LIN {X 0,Y 467.559,Z 249.866,A -85,B 0,C 180,E1 -7501.046,E2 -7501.046} C_VEL
LIN {X 0,Y 467.576,Z 249.863,A -85,B 0,C 180,E1 -7504.243,E2 -7504.243} C_VEL
LIN {X 0,Y 467.538,Z 249.871,A -85,B 0,C 180,E1 -7507.188,E2 -7507.188} C_VEL
LIN {X 0,Y 467.588,Z 249.861,A -85,B 0,C 180,E1 -7510.263,E2 -7510.263} C_VEL
LIN {X 0,Y 467.605,Z 249.859,A -85,B 0,C 180,E1 -7512.572,E2 -7512.572} C_VEL
LIN {X 0,Y 467.561,Z 249.864,A -85,B 0,C 180,E1 -7516.177,E2 -7516.177} C_VEL
LIN {X 0,Y 467.577,Z 249.864,A -85,B 0,C 180,E1 -7518.722,E2 -7518.722} C_VEL
LIN {X 0,Y 467.565,Z 249.869,A -85,B 0,C 180,E1 -7521.407,E2 -7521.407} C_VEL
LIN {X 0,Y 467.55,Z 249.865,A -85,B 0,C 180,E1 -7524.261,E2 -7524.261} C_VEL
LIN {X 0,Y 467.569,Z 249.868,A -85,B 0,C 180,E1 -7527.322,E2 -7527.322} C_VEL
LIN {X 0,Y 467.566,Z 249.867,A -85,B 0,C 180,E1 -7530.666,E2 -7530.666} C_VEL
LIN {X 0,Y 467.616,Z 249.862,A -85,B 0,C 180,E1 -7533.201,E2 -7533.201} C_VEL
LIN {X 0,Y 467.581,Z 249.864,A -85,B 0,C 180,E1 -7536.469,E2 -7536.469} C_VEL
LIN {X 0,Y 467.612,Z 249.858,A -85,B 0,C 180,E1 -7539.778,E2 -7539.778} C_VEL
LIN {X 0,Y 467.599,Z 249.863,A -85,B 0,C 180,E1 -7542.508,E2 -7542.508} C_VEL
LIN {X 0,Y 467.596,Z 249.862,A -85,B 0,C 180,E1 -7545.198,E2 -7545.198} C_VEL
LIN {X 0,Y 467.645,Z 249.854,A -85,B 0,C 180,E1 -7547.856,E2 -7547.856} C_VEL
LIN {X 0,Y 467.672,Z 249.851,A -85,B 0,C 180,E1 -7551.358,E2 -7551.358} C_VEL
LIN {X 0,Y 467.738,Z 249.843,A -85,B 0,C 180,E1 -7553.964,E2 -7553.964} C_VEL
LIN {X 0,Y 467.852,Z 249.828,A -85,B 0,C 180,E1 -7557.418,E2 -7557.418} C_VEL
LIN {X 0,Y 467.874,Z 249.827,A -85,B 0,C 180,E1 -7560.001,E2 -7560.001} C_VEL
LIN {X 0,Y 467.852,Z 249.834,A -85,B 0,C 180,E1 -7562.584,E2 -7562.584} C_VEL
LIN {X 0,Y 467.736,Z 249.846,A -85,B 0,C 180,E1 -7566.039,E2 -7566.039} C_VEL
LIN {X 0,Y 467.675,Z 249.854,A -85,B 0,C 180,E1 -7568.644,E2 -7568.644} C_VEL
LIN {X 0,Y 467.649,Z 249.86,A -85,B 0,C 180,E1 -7572.147,E2 -7572.147} C_VEL
LIN {X 0,Y 467.661,Z 249.856,A -85,B 0,C 180,E1 -7575.894,E2 -7575.894} C_VEL
LIN {X 0,Y 467.618,Z 249.857,A -85,B 0,C 180,E1 -7579.309,E2 -7579.309} C_VEL
LIN {X 0,Y 467.53,Z 249.876,A -85,B 0,C 180,E1 -7582.075,E2 -7582.075} C_VEL
LIN {X 0,Y 467.599,Z 249.859,A -85,B 0,C 180,E1 -7584.888,E2 -7584.888} C_VEL
LIN {X 0,Y 467.617,Z 249.862,A -85,B 0,C 180,E1 -7587.77,E2 -7587.77} C_VEL
LIN {X 0,Y 467.569,Z 249.863,A -85,B 0,C 180,E1 -7591.047,E2 -7591.047} C_VEL
LIN {X 0,Y 467.587,Z 249.864,A -85,B 0,C 180,E1 -7594.244,E2 -7594.244} C_VEL
LIN {X 0,Y 467.548,Z 249.867,A -85,B 0,C 180,E1 -7597.188,E2 -7597.188} C_VEL
LIN {X 0,Y 467.576,Z 249.864,A -85,B 0,C 180,E1 -7600.266,E2 -7600.266} C_VEL
LIN {X 0,Y 467.585,Z 249.861,A -85,B 0,C 180,E1 -7602.568,E2 -7602.568} C_VEL
LIN {X 0,Y 467.569,Z 249.864,A -85,B 0,C 180,E1 -7605.054,E2 -7605.054} C_VEL
LIN {X 0,Y 467.589,Z 249.866,A -85,B 0,C 180,E1 -7607.441,E2 -7607.441} C_VEL
LIN {X 0,Y 467.559,Z 249.865,A -85,B 0,C 180,E1 -7610.854,E2 -7610.854} C_VEL
LIN {X 0,Y 467.56,Z 249.865,A -85,B 0,C 180,E1 -7614.262,E2 -7614.262} C_VEL
LIN {X 0,Y 467.583,Z 249.868,A -85,B 0,C 180,E1 -7617.322,E2 -7617.322} C_VEL
LIN {X 0,Y 467.571,Z 249.869,A -85,B 0,C 180,E1 -7620.668,E2 -7620.668} C_VEL
LIN {X 0,Y 467.657,Z 250.033,A -85,B 0,C 180,E1 -7622.276,E2 -7622.276} C_VEL
LIN {X 0,Y 470.699,Z 264.33,A -85,B 0,C 180,E1 -7624.816,E2 -7624.816} C_VEL
LIN {X 0,Y 470.515,Z 271.163,A -85,B 0,C 180,E1 -7625.927,E2 -7625.927} C_VEL
LIN {X 0,Y 469.617,Z 290.074,A -85,B 0,C 180,E1 -7628.951,E2 -7628.951} C_VEL
LIN {X 0,Y 469.483,Z 293.151,A -85,B 0,C 180,E1 -7629.44,E2 -7629.44} C_VEL
LIN {X 0,Y 473.262,Z 315.105,A -85,B 0,C 180,E1 -7629.948,E2 -7629.948} C_VEL
LIN {X 0,Y 472.112,Z 431.405,A -85,B 0,C 180,E1 -7631.756,E2 -7631.756} C_VEL
LIN {X 0,Y 471.636,Z 446.004,A -85,B 0,C 180,E1 -7632.157,E2 -7632.157} C_VEL
LIN {X 0,Y 471.213,Z 458.569,A -85,B 0,C 180,E1 -7632.659,E2 -7632.659} C_VEL
LIN {X 0,Y 470.615,Z 471.376,A -85,B 0,C 180,E1 -7633.332,E2 -7633.332} C_VEL
LIN {X 0,Y 469.961,Z 483.799,A -85,B 0,C 180,E1 -7634.162,E2 -7634.162} C_VEL
LIN {X 0,Y 469.293,Z 495.623,A -85,B 0,C 180,E1 -7635.14,E2 -7635.14} C_VEL
LIN {X 0,Y 468.67,Z 505.453,A -85,B 0,C 180,E1 -7636.118,E2 -7636.118} C_VEL
LIN {X 0,Y 468.146,Z 515.918,A -85,B 0,C 180,E1 -7637.373,E2 -7637.373} C_VEL
LIN {X 0,Y 467.67,Z 525.293,A -85,B 0,C 180,E1 -7638.734,E2 -7638.734} C_VEL
LIN {X 0,Y 467.228,Z 533.88,A -85,B 0,C 180,E1 -7640.258,E2 -7640.258} C_VEL
LIN {X 0,Y 466.947,Z 540.8,A -85,B 0,C 180,E1 -7641.78,E2 -7641.78} C_VEL
LIN {X 0,Y 466.824,Z 545.573,A -85,B 0,C 180,E1 -7643.083,E2 -7643.083} C_VEL
LIN {X 0,Y 466.728,Z 550.51,A -85,B 0,C 180,E1 -7644.816,E2 -7644.816} C_VEL
LIN {X 0,Y 466.652,Z 553.941,A -85,B 0,C 180,E1 -7646.546,E2 -7646.546} C_VEL
LIN {X 0,Y 466.605,Z 555.971,A -85,B 0,C 180,E1 -7648.274,E2 -7648.274} C_VEL
LIN {X 0,Y 466.598,Z 556.648,A -85,B 0,C 180,E1 -7650,E2 -7650} C_VEL
LIN {X 0,Y 466.605,Z 555.983,A -85,B 0,C 180,E1 -7651.726,E2 -7651.726} C_VEL
LIN {X 0,Y 466.652,Z 553.966,A -85,B 0,C 180,E1 -7653.454,E2 -7653.454} C_VEL
LIN {X 0,Y 466.729,Z 550.553,A -85,B 0,C 180,E1 -7655.183,E2 -7655.183} C_VEL
LIN {X 0,Y 466.823,Z 545.641,A -85,B 0,C 180,E1 -7656.917,E2 -7656.917} C_VEL
LIN {X 0,Y 467.027,Z 539.091,A -85,B 0,C 180,E1 -7658.655,E2 -7658.655} C_VEL
LIN {X 0,Y 467.299,Z 531.81,A -85,B 0,C 180,E1 -7660.178,E2 -7660.178} C_VEL
LIN {X 0,Y 467.852,Z 522.814,A -85,B 0,C 180,E1 -7661.7,E2 -7661.7} C_VEL
LIN {X 0,Y 468.33,Z 513.378,A -85,B 0,C 180,E1 -7663.008,E2 -7663.008} C_VEL
LIN {X 0,Y 468.972,Z 501.875,A -85,B 0,C 180,E1 -7664.315,E2 -7664.315} C_VEL
LIN {X 0,Y 469.736,Z 490.184,A -85,B 0,C 180,E1 -7665.4,E2 -7665.4} C_VEL
LIN {X 0,Y 470.352,Z 478.783,A -85,B 0,C 180,E1 -7666.269,E2 -7666.269} C_VEL
LIN {X 0,Y 471.025,Z 466.302,A -85,B 0,C 180,E1 -7667.034,E2 -7667.034} C_VEL
LIN {X 0,Y 471.6,Z 452.42,A -85,B 0,C 180,E1 -7667.692,E2 -7667.692} C_VEL
LIN {X 0,Y 472.176,Z 437.842,A -85,B 0,C 180,E1 -7668.183,E2 -7668.183} C_VEL
LIN {X 0,Y 472.478,Z 423.654,A -85,B 0,C 180,E1 -7668.482,E2 -7668.482} C_VEL
LIN {X 0,Y 473.578,Z 314.653,A -85,B 0,C 180,E1 -7670.174,E2 -7670.174} C_VEL
LIN {X 0,Y 469.645,Z 292.953,A -85,B 0,C 180,E1 -7670.718,E2 -7670.718} C_VEL
LIN {X 0,Y 470.739,Z 273.148,A -85,B 0,C 180,E1 -7673.94,E2 -7673.94} C_VEL
LIN {X 0,Y 471.057,Z 265.779,A -85,B 0,C 180,E1 -7675.163,E2 -7675.163} C_VEL
LIN {X 0,Y 468.784,Z 254.744,A -85,B 0,C 180,E1 -7677.196,E2 -7677.196} C_VEL
LIN {X 0,Y 467.611,Z 249.864,A -85,B 0,C 180,E1 -7678.134,E2 -7678.134} C_VEL
LIN {X 0,Y 467.583,Z 249.868,A -85,B 0,C 180,E1 -7681.739,E2 -7681.739} C_VEL
LIN {X 0,Y 467.564,Z 249.871,A -85,B 0,C 180,E1 -7684.832,E2 -7684.832} C_VEL
LIN {X 0,Y 467.564,Z 249.867,A -85,B 0,C 180,E1 -7688.044,E2 -7688.044} C_VEL
LIN {X 0,Y 467.582,Z 249.861,A -85,B 0,C 180,E1 -7691.276,E2 -7691.276} C_VEL
LIN {X 0,Y 467.573,Z 249.867,A -85,B 0,C 180,E1 -7693.822,E2 -7693.822} C_VEL
LIN {X 0,Y 467.586,Z 249.863,A -85,B 0,C 180,E1 -7697.439,E2 -7697.439} C_VEL
LIN {X 0,Y 467.579,Z 249.864,A -85,B 0,C 180,E1 -7700.854,E2 -7700.854} C_VEL
LIN {X 0,Y 467.559,Z 249.858,A -85,B 0,C 180,E1 -7704.259,E2 -7704.259} C_VEL
LIN {X 0,Y 467.578,Z 249.864,A -85,B 0,C 180,E1 -7707.32,E2 -7707.32} C_VEL
LIN {X 0,Y 467.572,Z 249.864,A -85,B 0,C 180,E1 -7710.665,E2 -7710.665} C_VEL
LIN {X 0,Y 467.611,Z 249.858,A -85,B 0,C 180,E1 -7713.198,E2 -7713.198} C_VEL
LIN {X 0,Y 467.587,Z 249.861,A -85,B 0,C 180,E1 -7716.467,E2 -7716.467} C_VEL
LIN {X 0,Y 467.616,Z 249.86,A -85,B 0,C 180,E1 -7719.776,E2 -7719.776} C_VEL
LIN {X 0,Y 467.602,Z 249.86,A -85,B 0,C 180,E1 -7722.506,E2 -7722.506} C_VEL
LIN {X 0,Y 467.599,Z 249.861,A -85,B 0,C 180,E1 -7725.195,E2 -7725.195} C_VEL
LIN {X 0,Y 467.649,Z 249.853,A -85,B 0,C 180,E1 -7727.853,E2 -7727.853} C_VEL
LIN {X 0,Y 467.674,Z 249.856,A -85,B 0,C 180,E1 -7731.356,E2 -7731.356} C_VEL
LIN {X 0,Y 467.735,Z 249.845,A -85,B 0,C 180,E1 -7733.961,E2 -7733.961} C_VEL
LIN {X 0,Y 467.851,Z 249.831,A -85,B 0,C 180,E1 -7737.416,E2 -7737.416} C_VEL
LIN {X 0,Y 467.872,Z 249.826,A -85,B 0,C 180,E1 -7739.999,E2 -7739.999} C_VEL
LIN {X 0,Y 467.85,Z 249.828,A -85,B 0,C 180,E1 -7742.582,E2 -7742.582} C_VEL
LIN {X 0,Y 467.733,Z 249.841,A -85,B 0,C 180,E1 -7746.036,E2 -7746.036} C_VEL
LIN {X 0,Y 467.671,Z 249.854,A -85,B 0,C 180,E1 -7748.642,E2 -7748.642} C_VEL
LIN {X 0,Y 467.645,Z 249.855,A -85,B 0,C 180,E1 -7752.144,E2 -7752.144} C_VEL
LIN {X 0,Y 467.626,Z 249.857,A -85,B 0,C 180,E1 -7755.694,E2 -7755.694} C_VEL
LIN {X 0,Y 467.605,Z 249.865,A -85,B 0,C 180,E1 -7758.764,E2 -7758.764} C_VEL
LIN {X 0,Y 467.597,Z 249.863,A -85,B 0,C 180,E1 -7761.277,E2 -7761.277} C_VEL
LIN {X 0,Y 467.562,Z 249.863,A -85,B 0,C 180,E1 -7763.942,E2 -7763.942} C_VEL
LIN {X 0,Y 467.603,Z 249.864,A -85,B 0,C 180,E1 -7766.799,E2 -7766.799} C_VEL
LIN {X 0,Y 467.573,Z 249.861,A -85,B 0,C 180,E1 -7769.735,E2 -7769.735} C_VEL
LIN {X 0,Y 467.569,Z 249.87,A -85,B 0,C 180,E1 -7772.758,E2 -7772.758} C_VEL
LIN {X 0,Y 467.541,Z 249.864,A -85,B 0,C 180,E1 -7775.889,E2 -7775.889} C_VEL
LIN {X 0,Y 467.601,Z 249.859,A -85,B 0,C 180,E1 -7779.141,E2 -7779.141} C_VEL
LIN {X 0,Y 467.604,Z 249.863,A -85,B 0,C 180,E1 -7782.571,E2 -7782.571} C_VEL
LIN {X 0,Y 467.559,Z 249.872,A -85,B 0,C 180,E1 -7786.176,E2 -7786.176} C_VEL
LIN {X 0,Y 467.574,Z 249.866,A -85,B 0,C 180,E1 -7788.721,E2 -7788.721} C_VEL
LIN {X 0,Y 467.606,Z 249.923,A -85,B 0,C 180,E1 -7791.4,E2 -7791.4} C_VEL
LIN {X 0,Y 470.158,Z 262.256,A -85,B 0,C 180,E1 -7793.981,E2 -7793.981} C_VEL
LIN {X 0,Y 469.866,Z 269.478,A -85,B 0,C 180,E1 -7795.349,E2 -7795.349} C_VEL
LIN {X 0,Y 473.76,Z 287.231,A -85,B 0,C 180,E1 -7795.831,E2 -7795.831} C_VEL
LIN {X 0,Y 472.595,Z 401.54,A -85,B 0,C 180,E1 -7797.615,E2 -7797.615} C_VEL
LIN {X 0,Y 472.256,Z 405.426,A -85,B 0,C 180,E1 -7797.674,E2 -7797.674} C_VEL
LIN {X 0,Y 470.929,Z 411.156,A -85,B 0,C 180,E1 -7797.757,E2 -7797.757} C_VEL
LIN {X 0,Y 466.084,Z 425.092,A -85,B 0,C 180,E1 -7798.009,E2 -7798.009} C_VEL
LIN {X 0,Y 465.031,Z 431.625,A -85,B 0,C 180,E1 -7798.248,E2 -7798.248} C_VEL
LIN {X 0,Y 464.439,Z 444.396,A -85,B 0,C 180,E1 -7798.911,E2 -7798.911} C_VEL
LIN {X 0,Y 463.798,Z 456.799,A -85,B 0,C 180,E1 -7799.734,E2 -7799.734} C_VEL
LIN {X 0,Y 463.03,Z 468.474,A -85,B 0,C 180,E1 -7800.693,E2 -7800.693} C_VEL
LIN {X 0,Y 462.274,Z 480.207,A -85,B 0,C 180,E1 -7801.882,E2 -7801.882} C_VEL
LIN {X 0,Y 461.648,Z 489.89,A -85,B 0,C 180,E1 -7803.071,E2 -7803.071} C_VEL
LIN {X 0,Y 461.034,Z 499.712,A -85,B 0,C 180,E1 -7804.534,E2 -7804.534} C_VEL
LIN {X 0,Y 460.527,Z 507.999,A -85,B 0,C 180,E1 -7806.047,E2 -7806.047} C_VEL
LIN {X 0,Y 460.144,Z 514.68,A -85,B 0,C 180,E1 -7807.553,E2 -7807.553} C_VEL
LIN {X 0,Y 459.849,Z 520.148,A -85,B 0,C 180,E1 -7809.095,E2 -7809.095} C_VEL
LIN {X 0,Y 459.686,Z 524.788,A -85,B 0,C 180,E1 -7810.81,E2 -7810.81} C_VEL
LIN {X 0,Y 459.553,Z 527.485,A -85,B 0,C 180,E1 -7812.19,E2 -7812.19} C_VEL
LIN {X 0,Y 459.45,Z 529.765,A -85,B 0,C 180,E1 -7814.018,E2 -7814.018} C_VEL
LIN {X 0,Y 459.494,Z 530.362,A -85,B 0,C 180,E1 -7814.929,E2 -7814.929} C_VEL
LIN {X 0,Y 459.43,Z 530.506,A -85,B 0,C 180,E1 -7816.735,E2 -7816.735} C_VEL
LIN {X 0,Y 459.553,Z 529.261,A -85,B 0,C 180,E1 -7818.533,E2 -7818.533} C_VEL
LIN {X 0,Y 459.528,Z 526.622,A -85,B 0,C 180,E1 -7820.315,E2 -7820.315} C_VEL
LIN {X 0,Y 459.759,Z 522.522,A -85,B 0,C 180,E1 -7822.093,E2 -7822.093} C_VEL
LIN {X 0,Y 459.989,Z 516.886,A -85,B 0,C 180,E1 -7823.861,E2 -7823.861} C_VEL
LIN {X 0,Y 460.24,Z 510.554,A -85,B 0,C 180,E1 -7825.402,E2 -7825.402} C_VEL
LIN {X 0,Y 460.669,Z 502.693,A -85,B 0,C 180,E1 -7826.939,E2 -7826.939} C_VEL
LIN {X 0,Y 461.204,Z 494.486,A -85,B 0,C 180,E1 -7828.254,E2 -7828.254} C_VEL
LIN {X 0,Y 461.807,Z 484.641,A -85,B 0,C 180,E1 -7829.564,E2 -7829.564} C_VEL
LIN {X 0,Y 462.521,Z 473.711,A -85,B 0,C 180,E1 -7830.762,E2 -7830.762} C_VEL
LIN {X 0,Y 463.251,Z 461.53,A -85,B 0,C 180,E1 -7831.848,E2 -7831.848} C_VEL
LIN {X 0,Y 463.921,Z 449.502,A -85,B 0,C 180,E1 -7832.713,E2 -7832.713} C_VEL
LIN {X 0,Y 464.518,Z 436.222,A -85,B 0,C 180,E1 -7833.47,E2 -7833.47} C_VEL
LIN {X 0,Y 464.988,Z 423.124,A -85,B 0,C 180,E1 -7834.036,E2 -7834.036} C_VEL
LIN {X 0,Y 465.325,Z 408.995,A -85,B 0,C 180,E1 -7834.467,E2 -7834.467} C_VEL
LIN {X 0,Y 465.621,Z 388.412,A -85,B 0,C 180,E1 -7834.833,E2 -7834.833} C_VEL
LIN {X 0,Y 466.608,Z 287.767,A -85,B 0,C 180,E1 -7836.404,E2 -7836.404} C_VEL
LIN {X 0,Y 462.682,Z 269.347,A -85,B 0,C 180,E1 -7836.879,E2 -7836.879} C_VEL
LIN {X 0,Y 462.829,Z 261.896,A -85,B 0,C 180,E1 -7838.294,E2 -7838.294} C_VEL
LIN {X 0,Y 460.594,Z 250.738,A -85,B 0,C 180,E1 -7840.606,E2 -7840.606} C_VEL
LIN {X 0,Y 460.578,Z 250.738,A -85,B 0,C 180,E1 -7843.231,E2 -7843.231} C_VEL
LIN {X 0,Y 460.586,Z 250.739,A -85,B 0,C 180,E1 -7845.998,E2 -7845.998} C_VEL
LIN {X 0,Y 460.557,Z 250.737,A -85,B 0,C 180,E1 -7848.902,E2 -7848.902} C_VEL
LIN {X 0,Y 460.502,Z 250.748,A -85,B 0,C 180,E1 -7851.486,E2 -7851.486} C_VEL
LIN {X 0,Y 460.533,Z 250.741,A -85,B 0,C 180,E1 -7854.332,E2 -7854.332} C_VEL
LIN {X 0,Y 460.57,Z 250.738,A -85,B 0,C 180,E1 -7857.243,E2 -7857.243} C_VEL
LIN {X 0,Y 460.513,Z 250.743,A -85,B 0,C 180,E1 -7860.239,E2 -7860.239} C_VEL
LIN {X 0,Y 460.515,Z 250.747,A -85,B 0,C 180,E1 -7863.325,E2 -7863.325} C_VEL
LIN {X 0,Y 460.465,Z 250.748,A -85,B 0,C 180,E1 -7866.53,E2 -7866.53} C_VEL
LIN {X 0,Y 460.571,Z 250.737,A -85,B 0,C 180,E1 -7869.857,E2 -7869.857} C_VEL
LIN {X 0,Y 460.529,Z 250.742,A -85,B 0,C 180,E1 -7872.905,E2 -7872.905} C_VEL
LIN {X 0,Y 460.51,Z 250.744,A -85,B 0,C 180,E1 -7875.829,E2 -7875.829} C_VEL
LIN {X 0,Y 460.53,Z 250.744,A -85,B 0,C 180,E1 -7878.991,E2 -7878.991} C_VEL
LIN {X 0,Y 460.534,Z 250.747,A -85,B 0,C 180,E1 -7881.27,E2 -7881.27} C_VEL
LIN {X 0,Y 460.501,Z 250.745,A -85,B 0,C 180,E1 -7884.556,E2 -7884.556} C_VEL
LIN {X 0,Y 460.52,Z 250.742,A -85,B 0,C 180,E1 -7887.717,E2 -7887.717} C_VEL
LIN {X 0,Y 460.535,Z 250.744,A -85,B 0,C 180,E1 -7890.771,E2 -7890.771} C_VEL
LIN {X 0,Y 460.556,Z 250.737,A -85,B 0,C 180,E1 -7893.736,E2 -7893.736} C_VEL
LIN {X 0,Y 460.534,Z 250.743,A -85,B 0,C 180,E1 -7896.625,E2 -7896.625} C_VEL
LIN {X 0,Y 460.54,Z 250.74,A -85,B 0,C 180,E1 -7899.454,E2 -7899.454} C_VEL
LIN {X 0,Y 460.548,Z 250.739,A -85,B 0,C 180,E1 -7902.231,E2 -7902.231} C_VEL
LIN {X 0,Y 460.555,Z 250.742,A -85,B 0,C 180,E1 -7904.966,E2 -7904.966} C_VEL
LIN {X 0,Y 460.598,Z 250.731,A -85,B 0,C 180,E1 -7907.667,E2 -7907.667} C_VEL
LIN {X 0,Y 460.619,Z 250.73,A -85,B 0,C 180,E1 -7911.225,E2 -7911.225} C_VEL
LIN {X 0,Y 460.704,Z 250.719,A -85,B 0,C 180,E1 -7913.871,E2 -7913.871} C_VEL
LIN {X 0,Y 460.817,Z 250.704,A -85,B 0,C 180,E1 -7917.379,E2 -7917.379} C_VEL
LIN {X 0,Y 460.845,Z 250.703,A -85,B 0,C 180,E1 -7920.001,E2 -7920.001} C_VEL
LIN {X 0,Y 460.817,Z 250.71,A -85,B 0,C 180,E1 -7922.624,E2 -7922.624} C_VEL
LIN {X 0,Y 460.702,Z 250.723,A -85,B 0,C 180,E1 -7926.131,E2 -7926.131} C_VEL
LIN {X 0,Y 460.622,Z 250.731,A -85,B 0,C 180,E1 -7928.777,E2 -7928.777} C_VEL
LIN {X 0,Y 460.607,Z 250.736,A -85,B 0,C 180,E1 -7932.446,E2 -7932.446} C_VEL
LIN {X 0,Y 460.617,Z 250.735,A -85,B 0,C 180,E1 -7936.008,E2 -7936.008} C_VEL
LIN {X 0,Y 460.564,Z 250.738,A -85,B 0,C 180,E1 -7939.617,E2 -7939.617} C_VEL
LIN {X 0,Y 460.506,Z 250.746,A -85,B 0,C 180,E1 -7942.43,E2 -7942.43} C_VEL
LIN {X 0,Y 460.564,Z 250.741,A -85,B 0,C 180,E1 -7945.803,E2 -7945.803} C_VEL
LIN {X 0,Y 460.551,Z 250.742,A -85,B 0,C 180,E1 -7948.234,E2 -7948.234} C_VEL
LIN {X 0,Y 460.521,Z 250.742,A -85,B 0,C 180,E1 -7951.285,E2 -7951.285} C_VEL
LIN {X 0,Y 460.531,Z 250.741,A -85,B 0,C 180,E1 -7954.507,E2 -7954.507} C_VEL
LIN {X 0,Y 460.526,Z 250.746,A -85,B 0,C 180,E1 -7957.622,E2 -7957.622} C_VEL
LIN {X 0,Y 460.54,Z 250.741,A -85,B 0,C 180,E1 -7960.27,E2 -7960.27} C_VEL
LIN {X 0,Y 460.498,Z 250.748,A -85,B 0,C 180,E1 -7963.376,E2 -7963.376} C_VEL
LIN {X 0,Y 460.499,Z 250.744,A -85,B 0,C 180,E1 -7966.626,E2 -7966.626} C_VEL
LIN {X 0,Y 460.538,Z 250.745,A -85,B 0,C 180,E1 -7969.732,E2 -7969.732} C_VEL
LIN {X 0,Y 460.499,Z 250.744,A -85,B 0,C 180,E1 -7972.525,E2 -7972.525} C_VEL
LIN {X 0,Y 460.547,Z 250.746,A -85,B 0,C 180,E1 -7975.625,E2 -7975.625} C_VEL
LIN {X 0,Y 460.539,Z 250.746,A -85,B 0,C 180,E1 -7978.745,E2 -7978.745} C_VEL
LIN {X 0,Y 460.584,Z 250.79,A -85,B 0,C 180,E1 -7982.015,E2 -7982.015} C_VEL
LIN {X 0,Y 463.706,Z 265.39,A -85,B 0,C 180,E1 -7984.65,E2 -7984.65} C_VEL
LIN {X 0,Y 463.848,Z 268.795,A -85,B 0,C 180,E1 -7985.224,E2 -7985.224} C_VEL
LIN {X 0,Y 462.711,Z 289.716,A -85,B 0,C 180,E1 -7988.622,E2 -7988.622} C_VEL
LIN {X 0,Y 462.617,Z 293.272,A -85,B 0,C 180,E1 -7989.156,E2 -7989.156} C_VEL
LIN {X 0,Y 466.496,Z 315.37,A -85,B 0,C 180,E1 -7989.675,E2 -7989.675} C_VEL
LIN {X 0,Y 465.322,Z 431.416,A -85,B 0,C 180,E1 -7991.508,E2 -7991.508} C_VEL
LIN {X 0,Y 464.838,Z 445.946,A -85,B 0,C 180,E1 -7991.916,E2 -7991.916} C_VEL
LIN {X 0,Y 464.346,Z 459.301,A -85,B 0,C 180,E1 -7992.464,E2 -7992.464} C_VEL
LIN {X 0,Y 463.691,Z 472.438,A -85,B 0,C 180,E1 -7993.178,E2 -7993.178} C_VEL
LIN {X 0,Y 462.981,Z 484.771,A -85,B 0,C 180,E1 -7994.03,E2 -7994.03} C_VEL
LIN {X 0,Y 462.303,Z 496.406,A -85,B 0,C 180,E1 -7995.023,E2 -7995.023} C_VEL
LIN {X 0,Y 461.593,Z 507.067,A -85,B 0,C 180,E1 -7996.125,E2 -7996.125} C_VEL
LIN {X 0,Y 461.075,Z 517.705,A -85,B 0,C 180,E1 -7997.462,E2 -7997.462} C_VEL
LIN {X 0,Y 460.57,Z 526.369,A -85,B 0,C 180,E1 -7998.781,E2 -7998.781} C_VEL
LIN {X 0,Y 460.129,Z 534.721,A -85,B 0,C 180,E1 -8000.328,E2 -8000.328} C_VEL
LIN {X 0,Y 459.889,Z 540.542,A -85,B 0,C 180,E1 -8001.652,E2 -8001.652} C_VEL
LIN {X 0,Y 459.734,Z 545.327,A -85,B 0,C 180,E1 -8002.975,E2 -8002.975} C_VEL
LIN {X 0,Y 459.638,Z 550.277,A -85,B 0,C 180,E1 -8004.736,E2 -8004.736} C_VEL
LIN {X 0,Y 459.549,Z 553.719,A -85,B 0,C 180,E1 -8006.493,E2 -8006.493} C_VEL
LIN {X 0,Y 459.518,Z 555.76,A -85,B 0,C 180,E1 -8008.247,E2 -8008.247} C_VEL
LIN {X 0,Y 459.529,Z 556.448,A -85,B 0,C 180,E1 -8010,E2 -8010} C_VEL
LIN {X 0,Y 459.518,Z 555.794,A -85,B 0,C 180,E1 -8011.753,E2 -8011.753} C_VEL
LIN {X 0,Y 459.548,Z 553.787,A -85,B 0,C 180,E1 -8013.507,E2 -8013.507} C_VEL
LIN {X 0,Y 459.643,Z 550.383,A -85,B 0,C 180,E1 -8015.264,E2 -8015.264} C_VEL
LIN {X 0,Y 459.734,Z 545.48,A -85,B 0,C 180,E1 -8017.024,E2 -8017.024} C_VEL
LIN {X 0,Y 459.96,Z 538.94,A -85,B 0,C 180,E1 -8018.789,E2 -8018.789} C_VEL
LIN {X 0,Y 460.271,Z 531.677,A -85,B 0,C 180,E1 -8020.335,E2 -8020.335} C_VEL
LIN {X 0,Y 460.84,Z 522.715,A -85,B 0,C 180,E1 -8021.881,E2 -8021.881} C_VEL
LIN {X 0,Y 461.349,Z 513.323,A -85,B 0,C 180,E1 -8023.209,E2 -8023.209} C_VEL
LIN {X 0,Y 461.987,Z 502.94,A -85,B 0,C 180,E1 -8024.424,E2 -8024.424} C_VEL
LIN {X 0,Y 462.788,Z 491.511,A -85,B 0,C 180,E1 -8025.524,E2 -8025.524} C_VEL
LIN {X 0,Y 463.536,Z 478.872,A -85,B 0,C 180,E1 -8026.515,E2 -8026.515} C_VEL
LIN {X 0,Y 464.215,Z 467.054,A -85,B 0,C 180,E1 -8027.258,E2 -8027.258} C_VEL
LIN {X 0,Y 464.816,Z 453.354,A -85,B 0,C 180,E1 -8027.931,E2 -8027.931} C_VEL
LIN {X 0,Y 465.43,Z 439.139,A -85,B 0,C 180,E1 -8028.43,E2 -8028.43} C_VEL
LIN {X 0,Y 465.814,Z 424.647,A -85,B 0,C 180,E1 -8028.756,E2 -8028.756} C_VEL
LIN {X 0,Y 466.883,Z 315.127,A -85,B 0,C 180,E1 -8030.491,E2 -8030.491} C_VEL
LIN {X 0,Y 463.077,Z 294.302,A -85,B 0,C 180,E1 -8031.027,E2 -8031.027} C_VEL
LIN {X 0,Y 462.808,Z 292.65,A -85,B 0,C 180,E1 -8031.084,E2 -8031.084} C_VEL
LIN {X 0,Y 463.969,Z 273.005,A -85,B 0,C 180,E1 -8034.337,E2 -8034.337} C_VEL
LIN {X 0,Y 464.196,Z 267.202,A -85,B 0,C 180,E1 -8035.322,E2 -8035.322} C_VEL
LIN {X 0,Y 461.48,Z 254.587,A -85,B 0,C 180,E1 -8037.703,E2 -8037.703} C_VEL
LIN {X 0,Y 460.575,Z 250.741,A -85,B 0,C 180,E1 -8038.479,E2 -8038.479} C_VEL
LIN {X 0,Y 460.521,Z 250.748,A -85,B 0,C 180,E1 -8041.282,E2 -8041.282} C_VEL
LIN {X 0,Y 460.531,Z 250.747,A -85,B 0,C 180,E1 -8044.504,E2 -8044.504} C_VEL
LIN {X 0,Y 460.5,Z 250.745,A -85,B 0,C 180,E1 -8047.622,E2 -8047.622} C_VEL
LIN {X 0,Y 460.541,Z 250.742,A -85,B 0,C 180,E1 -8050.268,E2 -8050.268} C_VEL
LIN {X 0,Y 460.523,Z 250.743,A -85,B 0,C 180,E1 -8053.371,E2 -8053.371} C_VEL
LIN {X 0,Y 460.497,Z 250.748,A -85,B 0,C 180,E1 -8056.623,E2 -8056.623} C_VEL
LIN {X 0,Y 460.539,Z 250.743,A -85,B 0,C 180,E1 -8059.729,E2 -8059.729} C_VEL
LIN {X 0,Y 460.497,Z 250.744,A -85,B 0,C 180,E1 -8062.522,E2 -8062.522} C_VEL
LIN {X 0,Y 460.544,Z 250.734,A -85,B 0,C 180,E1 -8065.623,E2 -8065.623} C_VEL
LIN {X 0,Y 460.533,Z 250.737,A -85,B 0,C 180,E1 -8068.743,E2 -8068.743} C_VEL
LIN {X 0,Y 460.55,Z 250.742,A -85,B 0,C 180,E1 -8071.766,E2 -8071.766} C_VEL
LIN {X 0,Y 460.553,Z 250.738,A -85,B 0,C 180,E1 -8074.704,E2 -8074.704} C_VEL
LIN {X 0,Y 460.505,Z 250.748,A -85,B 0,C 180,E1 -8077.57,E2 -8077.57} C_VEL
LIN {X 0,Y 460.562,Z 250.736,A -85,B 0,C 180,E1 -8080.383,E2 -8080.383} C_VEL
LIN {X 0,Y 460.559,Z 250.739,A -85,B 0,C 180,E1 -8083.145,E2 -8083.145} C_VEL
LIN {X 0,Y 460.548,Z 250.743,A -85,B 0,C 180,E1 -8085.867,E2 -8085.867} C_VEL
LIN {X 0,Y 460.605,Z 250.727,A -85,B 0,C 180,E1 -8088.558,E2 -8088.558} C_VEL
LIN {X 0,Y 460.687,Z 250.717,A -85,B 0,C 180,E1 -8092.107,E2 -8092.107} C_VEL
LIN {X 0,Y 460.689,Z 250.722,A -85,B 0,C 180,E1 -8094.747,E2 -8094.747} C_VEL
LIN {X 0,Y 460.816,Z 250.707,A -85,B 0,C 180,E1 -8097.376,E2 -8097.376} C_VEL
LIN {X 0,Y 460.843,Z 250.701,A -85,B 0,C 180,E1 -8099.999,E2 -8099.999} C_VEL
LIN {X 0,Y 460.815,Z 250.705,A -85,B 0,C 180,E1 -8102.621,E2 -8102.621} C_VEL
LIN {X 0,Y 460.699,Z 250.717,A -85,B 0,C 180,E1 -8106.129,E2 -8106.129} C_VEL
LIN {X 0,Y 460.618,Z 250.734,A -85,B 0,C 180,E1 -8108.775,E2 -8108.775} C_VEL
LIN {X 0,Y 460.601,Z 250.734,A -85,B 0,C 180,E1 -8112.444,E2 -8112.444} C_VEL
LIN {X 0,Y 460.588,Z 250.734,A -85,B 0,C 180,E1 -8115.997,E2 -8115.997} C_VEL
LIN {X 0,Y 460.558,Z 250.744,A -85,B 0,C 180,E1 -8118.901,E2 -8118.901} C_VEL
LIN {X 0,Y 460.548,Z 250.74,A -85,B 0,C 180,E1 -8121.482,E2 -8121.482} C_VEL
LIN {X 0,Y 460.531,Z 250.741,A -85,B 0,C 180,E1 -8124.331,E2 -8124.331} C_VEL
LIN {X 0,Y 460.559,Z 250.739,A -85,B 0,C 180,E1 -8127.243,E2 -8127.243} C_VEL
LIN {X 0,Y 460.512,Z 250.741,A -85,B 0,C 180,E1 -8130.238,E2 -8130.238} C_VEL
LIN {X 0,Y 460.515,Z 250.744,A -85,B 0,C 180,E1 -8133.324,E2 -8133.324} C_VEL
LIN {X 0,Y 460.464,Z 250.753,A -85,B 0,C 180,E1 -8136.529,E2 -8136.529} C_VEL
LIN {X 0,Y 460.561,Z 250.737,A -85,B 0,C 180,E1 -8139.857,E2 -8139.857} C_VEL
LIN {X 0,Y 460.528,Z 250.745,A -85,B 0,C 180,E1 -8142.904,E2 -8142.904} C_VEL
LIN {X 0,Y 460.509,Z 250.747,A -85,B 0,C 180,E1 -8145.828,E2 -8145.828} C_VEL
LIN {X 0,Y 460.527,Z 250.744,A -85,B 0,C 180,E1 -8148.99,E2 -8148.99} C_VEL
LIN {X 0,Y 460.578,Z 250.798,A -85,B 0,C 180,E1 -8151.094,E2 -8151.094} C_VEL
LIN {X 0,Y 463.119,Z 263.055,A -85,B 0,C 180,E1 -8153.713,E2 -8153.713} C_VEL
LIN {X 0,Y 463.209,Z 267.162,A -85,B 0,C 180,E1 -8154.526,E2 -8154.526} C_VEL
LIN {X 0,Y 463.049,Z 269.623,A -85,B 0,C 180,E1 -8154.997,E2 -8154.997} C_VEL
LIN {X 0,Y 467.2,Z 288.578,A -85,B 0,C 180,E1 -8155.526,E2 -8155.526} C_VEL
LIN {X 0,Y 465.834,Z 406.782,A -85,B 0,C 180,E1 -8157.418,E2 -8157.418} C_VEL
LIN {X 0,Y 465.445,Z 420.776,A -85,B 0,C 180,E1 -8157.817,E2 -8157.817} C_VEL
LIN {X 0,Y 465.031,Z 431.625,A -85,B 0,C 180,E1 -8158.248,E2 -8158.248} C_VEL
LIN {X 0,Y 464.152,Z 437.177,A -85,B 0,C 180,E1 -8158.477,E2 -8158.477} C_VEL
LIN {X 0,Y 460.955,Z 446.079,A -85,B 0,C 180,E1 -8158.853,E2 -8158.853} C_VEL
LIN {X 0,Y 457.735,Z 454.693,A -85,B 0,C 180,E1 -8159.315,E2 -8159.315} C_VEL
LIN {X 0,Y 456.823,Z 459.74,A -85,B 0,C 180,E1 -8159.674,E2 -8159.674} C_VEL
LIN {X 0,Y 456.035,Z 471.505,A -85,B 0,C 180,E1 -8160.706,E2 -8160.706} C_VEL
LIN {X 0,Y 455.274,Z 481.988,A -85,B 0,C 180,E1 -8161.824,E2 -8161.824} C_VEL
LIN {X 0,Y 454.61,Z 492.022,A -85,B 0,C 180,E1 -8163.117,E2 -8163.117} C_VEL
LIN {X 0,Y 453.973,Z 501.266,A -85,B 0,C 180,E1 -8164.559,E2 -8164.559} C_VEL
LIN {X 0,Y 453.45,Z 509.431,A -85,B 0,C 180,E1 -8166.121,E2 -8166.121} C_VEL
LIN {X 0,Y 453.049,Z 515.927,A -85,B 0,C 180,E1 -8167.663,E2 -8167.663} C_VEL
LIN {X 0,Y 452.77,Z 520.725,A -85,B 0,C 180,E1 -8169.084,E2 -8169.084} C_VEL
LIN {X 0,Y 452.614,Z 524.496,A -85,B 0,C 180,E1 -8170.498,E2 -8170.498} C_VEL
LIN {X 0,Y 452.483,Z 527.352,A -85,B 0,C 180,E1 -8171.903,E2 -8171.903} C_VEL
LIN {X 0,Y 452.358,Z 529.782,A -85,B 0,C 180,E1 -8173.761,E2 -8173.761} C_VEL
LIN {X 0,Y 452.411,Z 530.453,A -85,B 0,C 180,E1 -8174.688,E2 -8174.688} C_VEL
LIN {X 0,Y 452.342,Z 530.743,A -85,B 0,C 180,E1 -8176.524,E2 -8176.524} C_VEL
LIN {X 0,Y 452.454,Z 529.646,A -85,B 0,C 180,E1 -8178.351,E2 -8178.351} C_VEL
LIN {X 0,Y 452.433,Z 527.183,A -85,B 0,C 180,E1 -8180.162,E2 -8180.162} C_VEL
LIN {X 0,Y 452.659,Z 523.273,A -85,B 0,C 180,E1 -8181.968,E2 -8181.968} C_VEL
LIN {X 0,Y 452.895,Z 517.796,A -85,B 0,C 180,E1 -8183.764,E2 -8183.764} C_VEL
LIN {X 0,Y 453.117,Z 512.626,A -85,B 0,C 180,E1 -8185.107,E2 -8185.107} C_VEL
LIN {X 0,Y 453.511,Z 505.185,A -85,B 0,C 180,E1 -8186.669,E2 -8186.669} C_VEL
LIN {X 0,Y 454.027,Z 497.445,A -85,B 0,C 180,E1 -8188.004,E2 -8188.004} C_VEL
LIN {X 0,Y 454.639,Z 488.141,A -85,B 0,C 180,E1 -8189.336,E2 -8189.336} C_VEL
LIN {X 0,Y 455.331,Z 477.871,A -85,B 0,C 180,E1 -8190.553,E2 -8190.553} C_VEL
LIN {X 0,Y 456.09,Z 466.565,A -85,B 0,C 180,E1 -8191.656,E2 -8191.656} C_VEL
LIN {X 0,Y 456.836,Z 454.086,A -85,B 0,C 180,E1 -8192.645,E2 -8192.645} C_VEL
LIN {X 0,Y 457.448,Z 442.027,A -85,B 0,C 180,E1 -8193.413,E2 -8193.413} C_VEL
LIN {X 0,Y 458.03,Z 427.994,A -85,B 0,C 180,E1 -8194.103,E2 -8194.103} C_VEL
LIN {X 0,Y 458.462,Z 414.254,A -85,B 0,C 180,E1 -8194.589,E2 -8194.589} C_VEL
LIN {X 0,Y 458.753,Z 399.824,A -85,B 0,C 180,E1 -8194.916,E2 -8194.916} C_VEL
LIN {X 0,Y 459.919,Z 288.821,A -85,B 0,C 180,E1 -8196.672,E2 -8196.672} C_VEL
LIN {X 0,Y 455.756,Z 269.446,A -85,B 0,C 180,E1 -8197.198,E2 -8197.198} C_VEL
LIN {X 0,Y 455.879,Z 263.086,A -85,B 0,C 180,E1 -8198.421,E2 -8198.421} C_VEL
LIN {X 0,Y 453.547,Z 251.615,A -85,B 0,C 180,E1 -8200.829,E2 -8200.829} C_VEL
LIN {X 0,Y 453.524,Z 251.617,A -85,B 0,C 180,E1 -8203.441,E2 -8203.441} C_VEL
LIN {X 0,Y 453.531,Z 251.615,A -85,B 0,C 180,E1 -8206.196,E2 -8206.196} C_VEL
LIN {X 0,Y 453.506,Z 251.615,A -85,B 0,C 180,E1 -8209.041,E2 -8209.041} C_VEL
LIN {X 0,Y 453.463,Z 251.627,A -85,B 0,C 180,E1 -8211.836,E2 -8211.836} C_VEL
LIN {X 0,Y 453.511,Z 251.614,A -85,B 0,C 180,E1 -8214.734,E2 -8214.734} C_VEL
LIN {X 0,Y 453.525,Z 251.616,A -85,B 0,C 180,E1 -8217.962,E2 -8217.962} C_VEL
LIN {X 0,Y 453.469,Z 251.62,A -85,B 0,C 180,E1 -8220.759,E2 -8220.759} C_VEL
LIN {X 0,Y 453.464,Z 251.623,A -85,B 0,C 180,E1 -8223.913,E2 -8223.913} C_VEL
LIN {X 0,Y 453.458,Z 251.625,A -85,B 0,C 180,E1 -8227.188,E2 -8227.188} C_VEL
LIN {X 0,Y 453.523,Z 251.62,A -85,B 0,C 180,E1 -8229.445,E2 -8229.445} C_VEL
LIN {X 0,Y 453.479,Z 251.622,A -85,B 0,C 180,E1 -8232.992,E2 -8232.992} C_VEL
LIN {X 0,Y 453.463,Z 251.622,A -85,B 0,C 180,E1 -8235.781,E2 -8235.781} C_VEL
LIN {X 0,Y 453.483,Z 251.618,A -85,B 0,C 180,E1 -8238.212,E2 -8238.212} C_VEL
LIN {X 0,Y 453.519,Z 251.616,A -85,B 0,C 180,E1 -8240.788,E2 -8240.788} C_VEL
LIN {X 0,Y 453.444,Z 251.623,A -85,B 0,C 180,E1 -8243.918,E2 -8243.918} C_VEL
LIN {X 0,Y 453.47,Z 251.627,A -85,B 0,C 180,E1 -8247.152,E2 -8247.152} C_VEL
LIN {X 0,Y 453.502,Z 251.616,A -85,B 0,C 180,E1 -8250.272,E2 -8250.272} C_VEL
LIN {X 0,Y 453.502,Z 251.619,A -85,B 0,C 180,E1 -8253.295,E2 -8253.295} C_VEL
LIN {X 0,Y 453.492,Z 251.617,A -85,B 0,C 180,E1 -8256.24,E2 -8256.24} C_VEL
LIN {X 0,Y 453.472,Z 251.624,A -85,B 0,C 180,E1 -8259.119,E2 -8259.119} C_VEL
LIN {X 0,Y 453.501,Z 251.616,A -85,B 0,C 180,E1 -8261.946,E2 -8261.946} C_VEL
LIN {X 0,Y 453.529,Z 251.62,A -85,B 0,C 180,E1 -8264.727,E2 -8264.727} C_VEL
LIN {X 0,Y 453.553,Z 251.609,A -85,B 0,C 180,E1 -8267.472,E2 -8267.472} C_VEL
LIN {X 0,Y 453.583,Z 251.608,A -85,B 0,C 180,E1 -8271.088,E2 -8271.088} C_VEL
LIN {X 0,Y 453.671,Z 251.595,A -85,B 0,C 180,E1 -8273.776,E2 -8273.776} C_VEL
LIN {X 0,Y 453.758,Z 251.584,A -85,B 0,C 180,E1 -8277.338,E2 -8277.338} C_VEL
LIN {X 0,Y 453.815,Z 251.578,A -85,B 0,C 180,E1 -8280.001,E2 -8280.001} C_VEL
LIN {X 0,Y 453.758,Z 251.588,A -85,B 0,C 180,E1 -8282.664,E2 -8282.664} C_VEL
LIN {X 0,Y 453.67,Z 251.6,A -85,B 0,C 180,E1 -8286.227,E2 -8286.227} C_VEL
LIN {X 0,Y 453.586,Z 251.606,A -85,B 0,C 180,E1 -8288.915,E2 -8288.915} C_VEL
LIN {X 0,Y 453.557,Z 251.613,A -85,B 0,C 180,E1 -8292.53,E2 -8292.53} C_VEL
LIN {X 0,Y 453.551,Z 251.617,A -85,B 0,C 180,E1 -8296.197,E2 -8296.197} C_VEL
LIN {X 0,Y 453.515,Z 251.614,A -85,B 0,C 180,E1 -8299.042,E2 -8299.042} C_VEL
LIN {X 0,Y 453.472,Z 251.624,A -85,B 0,C 180,E1 -8301.837,E2 -8301.837} C_VEL
LIN {X 0,Y 453.51,Z 251.615,A -85,B 0,C 180,E1 -8304.736,E2 -8304.736} C_VEL
LIN {X 0,Y 453.53,Z 251.62,A -85,B 0,C 180,E1 -8307.961,E2 -8307.961} C_VEL
LIN {X 0,Y 453.48,Z 251.618,A -85,B 0,C 180,E1 -8310.76,E2 -8310.76} C_VEL
LIN {X 0,Y 453.475,Z 251.626,A -85,B 0,C 180,E1 -8313.914,E2 -8313.914} C_VEL
LIN {X 0,Y 453.468,Z 251.621,A -85,B 0,C 180,E1 -8317.189,E2 -8317.189} C_VEL
LIN {X 0,Y 453.515,Z 251.618,A -85,B 0,C 180,E1 -8319.448,E2 -8319.448} C_VEL
LIN {X 0,Y 453.462,Z 251.621,A -85,B 0,C 180,E1 -8322.996,E2 -8322.996} C_VEL
LIN {X 0,Y 453.465,Z 251.626,A -85,B 0,C 180,E1 -8325.78,E2 -8325.78} C_VEL
LIN {X 0,Y 453.479,Z 251.62,A -85,B 0,C 180,E1 -8328.21,E2 -8328.21} C_VEL
LIN {X 0,Y 453.471,Z 251.62,A -85,B 0,C 180,E1 -8330.798,E2 -8330.798} C_VEL
LIN {X 0,Y 453.454,Z 251.624,A -85,B 0,C 180,E1 -8333.918,E2 -8333.918} C_VEL
LIN {X 0,Y 453.484,Z 251.622,A -85,B 0,C 180,E1 -8337.152,E2 -8337.152} C_VEL
LIN {X 0,Y 453.476,Z 251.625,A -85,B 0,C 180,E1 -8340.269,E2 -8340.269} C_VEL
LIN {X 0,Y 453.554,Z 251.737,A -85,B 0,C 180,E1 -8341.783,E2 -8341.783} C_VEL
LIN {X 0,Y 456.924,Z 267.651,A -85,B 0,C 180,E1 -8344.696,E2 -8344.696} C_VEL
LIN {X 0,Y 456.157,Z 283.626,A -85,B 0,C 180,E1 -8347.346,E2 -8347.346} C_VEL
LIN {X 0,Y 455.661,Z 292.77,A -85,B 0,C 180,E1 -8348.844,E2 -8348.844} C_VEL
LIN {X 0,Y 459.794,Z 316.776,A -85,B 0,C 180,E1 -8349.418,E2 -8349.418} C_VEL
LIN {X 0,Y 458.546,Z 430.216,A -85,B 0,C 180,E1 -8351.225,E2 -8351.225} C_VEL
LIN {X 0,Y 458.077,Z 444.354,A -85,B 0,C 180,E1 -8351.611,E2 -8351.611} C_VEL
LIN {X 0,Y 457.523,Z 458.002,A -85,B 0,C 180,E1 -8352.162,E2 -8352.162} C_VEL
LIN {X 0,Y 456.847,Z 472.027,A -85,B 0,C 180,E1 -8352.929,E2 -8352.929} C_VEL
LIN {X 0,Y 456.108,Z 484.278,A -85,B 0,C 180,E1 -8353.783,E2 -8353.783} C_VEL
LIN {X 0,Y 455.397,Z 495.965,A -85,B 0,C 180,E1 -8354.79,E2 -8354.79} C_VEL
LIN {X 0,Y 454.632,Z 506.666,A -85,B 0,C 180,E1 -8355.909,E2 -8355.909} C_VEL
LIN {X 0,Y 454.073,Z 516.773,A -85,B 0,C 180,E1 -8357.188,E2 -8357.188} C_VEL
LIN {X 0,Y 453.553,Z 526.039,A -85,B 0,C 180,E1 -8358.605,E2 -8358.605} C_VEL
LIN {X 0,Y 453.061,Z 534.428,A -85,B 0,C 180,E1 -8360.175,E2 -8360.175} C_VEL
LIN {X 0,Y 452.814,Z 540.269,A -85,B 0,C 180,E1 -8361.521,E2 -8361.521} C_VEL
LIN {X 0,Y 452.658,Z 545.075,A -85,B 0,C 180,E1 -8362.865,E2 -8362.865} C_VEL
LIN {X 0,Y 452.549,Z 550.042,A -85,B 0,C 180,E1 -8364.654,E2 -8364.654} C_VEL
LIN {X 0,Y 452.448,Z 553.497,A -85,B 0,C 180,E1 -8366.438,E2 -8366.438} C_VEL
LIN {X 0,Y 452.501,Z 554.695,A -85,B 0,C 180,E1 -8367.329,E2 -8367.329} C_VEL
LIN {X 0,Y 452.427,Z 556.066,A -85,B 0,C 180,E1 -8369.11,E2 -8369.11} C_VEL
LIN {X 0,Y 452.427,Z 556.093,A -85,B 0,C 180,E1 -8370.89,E2 -8370.89} C_VEL
LIN {X 0,Y 452.501,Z 554.78,A -85,B 0,C 180,E1 -8372.67,E2 -8372.67} C_VEL
LIN {X 0,Y 452.472,Z 552.093,A -85,B 0,C 180,E1 -8374.454,E2 -8374.454} C_VEL
LIN {X 0,Y 452.585,Z 547.971,A -85,B 0,C 180,E1 -8376.24,E2 -8376.24} C_VEL
LIN {X 0,Y 452.742,Z 542.291,A -85,B 0,C 180,E1 -8378.031,E2 -8378.031} C_VEL
LIN {X 0,Y 453.049,Z 535.898,A -85,B 0,C 180,E1 -8379.599,E2 -8379.599} C_VEL
LIN {X 0,Y 453.525,Z 527.963,A -85,B 0,C 180,E1 -8381.169,E2 -8381.169} C_VEL
LIN {X 0,Y 454.033,Z 518.945,A -85,B 0,C 180,E1 -8382.627,E2 -8382.627} C_VEL
LIN {X 0,Y 454.649,Z 509.717,A -85,B 0,C 180,E1 -8383.863,E2 -8383.863} C_VEL
LIN {X 0,Y 455.39,Z 498.656,A -85,B 0,C 180,E1 -8385.095,E2 -8385.095} C_VEL
LIN {X 0,Y 456.291,Z 486.327,A -85,B 0,C 180,E1 -8386.21,E2 -8386.21} C_VEL
LIN {X 0,Y 457.071,Z 473.268,A -85,B 0,C 180,E1 -8387.159,E2 -8387.159} C_VEL
LIN {X 0,Y 457.856,Z 459.503,A -85,B 0,C 180,E1 -8387.936,E2 -8387.936} C_VEL
LIN {X 0,Y 458.493,Z 445.726,A -85,B 0,C 180,E1 -8388.516,E2 -8388.516} C_VEL
LIN {X 0,Y 458.975,Z 431.47,A -85,B 0,C 180,E1 -8388.931,E2 -8388.931} C_VEL
LIN {X 0,Y 459.763,Z 372.166,A -85,B 0,C 180,E1 -8389.904,E2 -8389.904} C_VEL
LIN {X 0,Y 460.281,Z 315.903,A -85,B 0,C 180,E1 -8390.813,E2 -8390.813} C_VEL
LIN {X 0,Y 456.68,Z 296.173,A -85,B 0,C 180,E1 -8391.333,E2 -8391.333} C_VEL
LIN {X 0,Y 455.972,Z 292.451,A -85,B 0,C 180,E1 -8391.449,E2 -8391.449} C_VEL
LIN {X 0,Y 457.235,Z 272.707,A -85,B 0,C 180,E1 -8394.779,E2 -8394.779} C_VEL
LIN {X 0,Y 457.304,Z 268.641,A -85,B 0,C 180,E1 -8395.487,E2 -8395.487} C_VEL
LIN {X 0,Y 454.946,Z 257.583,A -85,B 0,C 180,E1 -8397.608,E2 -8397.608} C_VEL
LIN {X 0,Y 453.509,Z 251.619,A -85,B 0,C 180,E1 -8398.838,E2 -8398.838} C_VEL
LIN {X 0,Y 453.465,Z 251.628,A -85,B 0,C 180,E1 -8401.798,E2 -8401.798} C_VEL
LIN {X 0,Y 453.48,Z 251.625,A -85,B 0,C 180,E1 -8404.988,E2 -8404.988} C_VEL
LIN {X 0,Y 453.463,Z 251.626,A -85,B 0,C 180,E1 -8408.311,E2 -8408.311} C_VEL
LIN {X 0,Y 453.494,Z 251.617,A -85,B 0,C 180,E1 -8410.608,E2 -8410.608} C_VEL
LIN {X 0,Y 453.48,Z 251.62,A -85,B 0,C 180,E1 -8413.246,E2 -8413.246} C_VEL
LIN {X 0,Y 453.464,Z 251.624,A -85,B 0,C 180,E1 -8415.778,E2 -8415.778} C_VEL
LIN {X 0,Y 453.477,Z 251.624,A -85,B 0,C 180,E1 -8418.208,E2 -8418.208} C_VEL
LIN {X 0,Y 453.491,Z 251.619,A -85,B 0,C 180,E1 -8420.792,E2 -8420.792} C_VEL
LIN {X 0,Y 453.453,Z 251.615,A -85,B 0,C 180,E1 -8423.916,E2 -8423.916} C_VEL
LIN {X 0,Y 453.479,Z 251.619,A -85,B 0,C 180,E1 -8427.15,E2 -8427.15} C_VEL
LIN {X 0,Y 453.51,Z 251.619,A -85,B 0,C 180,E1 -8430.27,E2 -8430.27} C_VEL
LIN {X 0,Y 453.501,Z 251.616,A -85,B 0,C 180,E1 -8433.293,E2 -8433.293} C_VEL
LIN {X 0,Y 453.498,Z 251.618,A -85,B 0,C 180,E1 -8436.238,E2 -8436.238} C_VEL
LIN {X 0,Y 453.476,Z 251.62,A -85,B 0,C 180,E1 -8439.116,E2 -8439.116} C_VEL
LIN {X 0,Y 453.505,Z 251.62,A -85,B 0,C 180,E1 -8441.943,E2 -8441.943} C_VEL
LIN {X 0,Y 453.532,Z 251.61,A -85,B 0,C 180,E1 -8444.725,E2 -8444.725} C_VEL
LIN {X 0,Y 453.554,Z 251.605,A -85,B 0,C 180,E1 -8448.378,E2 -8448.378} C_VEL
LIN {X 0,Y 453.644,Z 251.595,A -85,B 0,C 180,E1 -8451.984,E2 -8451.984} C_VEL
LIN {X 0,Y 453.663,Z 251.597,A -85,B 0,C 180,E1 -8454.666,E2 -8454.666} C_VEL
LIN {X 0,Y 453.756,Z 251.585,A -85,B 0,C 180,E1 -8457.336,E2 -8457.336} C_VEL
LIN {X 0,Y 453.814,Z 251.577,A -85,B 0,C 180,E1 -8459.999,E2 -8459.999} C_VEL
LIN {X 0,Y 453.756,Z 251.584,A -85,B 0,C 180,E1 -8462.662,E2 -8462.662} C_VEL
LIN {X 0,Y 453.666,Z 251.593,A -85,B 0,C 180,E1 -8466.224,E2 -8466.224} C_VEL
LIN {X 0,Y 453.582,Z 251.611,A -85,B 0,C 180,E1 -8468.912,E2 -8468.912} C_VEL
LIN {X 0,Y 453.552,Z 251.613,A -85,B 0,C 180,E1 -8472.528,E2 -8472.528} C_VEL
LIN {X 0,Y 453.532,Z 251.613,A -85,B 0,C 180,E1 -8476.195,E2 -8476.195} C_VEL
LIN {X 0,Y 453.508,Z 251.621,A -85,B 0,C 180,E1 -8479.04,E2 -8479.04} C_VEL
LIN {X 0,Y 453.485,Z 251.619,A -85,B 0,C 180,E1 -8481.834,E2 -8481.834} C_VEL
LIN {X 0,Y 453.502,Z 251.62,A -85,B 0,C 180,E1 -8484.733,E2 -8484.733} C_VEL
LIN {X 0,Y 453.52,Z 251.615,A -85,B 0,C 180,E1 -8487.959,E2 -8487.959} C_VEL
LIN {X 0,Y 453.469,Z 251.615,A -85,B 0,C 180,E1 -8490.758,E2 -8490.758} C_VEL
LIN {X 0,Y 453.463,Z 251.623,A -85,B 0,C 180,E1 -8493.912,E2 -8493.912} C_VEL
LIN {X 0,Y 453.457,Z 251.625,A -85,B 0,C 180,E1 -8497.187,E2 -8497.187} C_VEL
LIN {X 0,Y 453.517,Z 251.613,A -85,B 0,C 180,E1 -8499.445,E2 -8499.445} C_VEL
LIN {X 0,Y 453.477,Z 251.623,A -85,B 0,C 180,E1 -8502.991,E2 -8502.991} C_VEL
LIN {X 0,Y 453.462,Z 251.625,A -85,B 0,C 180,E1 -8505.78,E2 -8505.78} C_VEL
LIN {X 0,Y 453.481,Z 251.625,A -85,B 0,C 180,E1 -8508.211,E2 -8508.211} C_VEL
LIN {X 0,Y 453.534,Z 251.716,A -85,B 0,C 180,E1 -8510.784,E2 -8510.784} C_VEL
LIN {X 0,Y 455.95,Z 263.124,A -85,B 0,C 180,E1 -8513.273,E2 -8513.273} C_VEL
LIN {X 0,Y 456.404,Z 267.551,A -85,B 0,C 180,E1 -8514.188,E2 -8514.188} C_VEL
LIN {X 0,Y 456.287,Z 269.975,A -85,B 0,C 180,E1 -8514.638,E2 -8514.638} C_VEL
LIN {X 0,Y 460.485,Z 288.515,A -85,B 0,C 180,E1 -8515.177,E2 -8515.177} C_VEL
LIN {X 0,Y 460.561,Z 299.284,A -85,B 0,C 180,E1 -8515.361,E2 -8515.361} C_VEL
LIN {X 0,Y 459.225,Z 406.215,A -85,B 0,C 180,E1 -8517.091,E2 -8517.091} C_VEL
LIN {X 0,Y 458.826,Z 420.163,A -85,B 0,C 180,E1 -8517.484,E2 -8517.484} C_VEL
LIN {X 0,Y 458.255,Z 433.992,A -85,B 0,C 180,E1 -8518.056,E2 -8518.056} C_VEL
LIN {X 0,Y 457.603,Z 447.074,A -85,B 0,C 180,E1 -8518.78,E2 -8518.78} C_VEL
LIN {X 0,Y 456.823,Z 459.74,A -85,B 0,C 180,E1 -8519.674,E2 -8519.674} C_VEL
LIN {X 0,Y 455.905,Z 464.738,A -85,B 0,C 180,E1 -8520.058,E2 -8520.058} C_VEL
LIN {X 0,Y 452.617,Z 472.694,A -85,B 0,C 180,E1 -8520.677,E2 -8520.677} C_VEL
LIN {X 0,Y 449.255,Z 480.269,A -85,B 0,C 180,E1 -8521.369,E2 -8521.369} C_VEL
LIN {X 0,Y 448.235,Z 484.609,A -85,B 0,C 180,E1 -8521.863,E2 -8521.863} C_VEL
LIN {X 0,Y 447.597,Z 493.774,A -85,B 0,C 180,E1 -8523.107,E2 -8523.107} C_VEL
LIN {X 0,Y 446.905,Z 502.997,A -85,B 0,C 180,E1 -8524.626,E2 -8524.626} C_VEL
LIN {X 0,Y 446.448,Z 509.562,A -85,B 0,C 180,E1 -8525.924,E2 -8525.924} C_VEL
LIN {X 0,Y 446.056,Z 515.302,A -85,B 0,C 180,E1 -8527.294,E2 -8527.294} C_VEL
LIN {X 0,Y 445.751,Z 520.268,A -85,B 0,C 180,E1 -8528.739,E2 -8528.739} C_VEL
LIN {X 0,Y 445.577,Z 524.208,A -85,B 0,C 180,E1 -8530.178,E2 -8530.178} C_VEL
LIN {X 0,Y 445.427,Z 527.211,A -85,B 0,C 180,E1 -8531.606,E2 -8531.606} C_VEL
LIN {X 0,Y 445.268,Z 529.802,A -85,B 0,C 180,E1 -8533.495,E2 -8533.495} C_VEL
LIN {X 0,Y 445.311,Z 530.546,A -85,B 0,C 180,E1 -8534.437,E2 -8534.437} C_VEL
LIN {X 0,Y 445.254,Z 530.98,A -85,B 0,C 180,E1 -8536.305,E2 -8536.305} C_VEL
LIN {X 0,Y 445.369,Z 530.024,A -85,B 0,C 180,E1 -8538.163,E2 -8538.163} C_VEL
LIN {X 0,Y 445.346,Z 527.702,A -85,B 0,C 180,E1 -8540.004,E2 -8540.004} C_VEL
LIN {X 0,Y 445.558,Z 523.956,A -85,B 0,C 180,E1 -8541.839,E2 -8541.839} C_VEL
LIN {X 0,Y 445.804,Z 518.697,A -85,B 0,C 180,E1 -8543.665,E2 -8543.665} C_VEL
LIN {X 0,Y 446.016,Z 513.624,A -85,B 0,C 180,E1 -8545.028,E2 -8545.028} C_VEL
LIN {X 0,Y 446.436,Z 506.396,A -85,B 0,C 180,E1 -8546.616,E2 -8546.616} C_VEL
LIN {X 0,Y 447.036,Z 497.464,A -85,B 0,C 180,E1 -8548.198,E2 -8548.198} C_VEL
LIN {X 0,Y 447.71,Z 488.104,A -85,B 0,C 180,E1 -8549.55,E2 -8549.55} C_VEL
LIN {X 0,Y 448.478,Z 476.724,A -85,B 0,C 180,E1 -8550.898,E2 -8550.898} C_VEL
LIN {X 0,Y 449.29,Z 465.123,A -85,B 0,C 180,E1 -8552.017,E2 -8552.017} C_VEL
LIN {X 0,Y 450.086,Z 452.259,A -85,B 0,C 180,E1 -8553.021,E2 -8553.021} C_VEL
LIN {X 0,Y 450.722,Z 439.671,A -85,B 0,C 180,E1 -8553.8,E2 -8553.8} C_VEL
LIN {X 0,Y 451.356,Z 425.522,A -85,B 0,C 180,E1 -8554.465,E2 -8554.465} C_VEL
LIN {X 0,Y 451.737,Z 411.253,A -85,B 0,C 180,E1 -8554.937,E2 -8554.937} C_VEL
LIN {X 0,Y 452.016,Z 396.199,A -85,B 0,C 180,E1 -8555.241,E2 -8555.241} C_VEL
LIN {X 0,Y 453.25,Z 290.119,A -85,B 0,C 180,E1 -8556.941,E2 -8556.941} C_VEL
LIN {X 0,Y 448.85,Z 269.769,A -85,B 0,C 180,E1 -8557.478,E2 -8557.478} C_VEL
LIN {X 0,Y 449.071,Z 265.402,A -85,B 0,C 180,E1 -8558.323,E2 -8558.323} C_VEL
LIN {X 0,Y 446.545,Z 252.488,A -85,B 0,C 180,E1 -8561.059,E2 -8561.059} C_VEL
LIN {X 0,Y 446.473,Z 252.497,A -85,B 0,C 180,E1 -8563.657,E2 -8563.657} C_VEL
LIN {X 0,Y 446.476,Z 252.492,A -85,B 0,C 180,E1 -8566.459,E2 -8566.459} C_VEL
LIN {X 0,Y 446.455,Z 252.495,A -85,B 0,C 180,E1 -8569.303,E2 -8569.303} C_VEL
LIN {X 0,Y 446.404,Z 252.502,A -85,B 0,C 180,E1 -8572.2,E2 -8572.2} C_VEL
LIN {X 0,Y 446.457,Z 252.495,A -85,B 0,C 180,E1 -8575.152,E2 -8575.152} C_VEL
LIN {X 0,Y 446.47,Z 252.493,A -85,B 0,C 180,E1 -8578.179,E2 -8578.179} C_VEL
LIN {X 0,Y 446.417,Z 252.502,A -85,B 0,C 180,E1 -8581.3,E2 -8581.3} C_VEL
LIN {X 0,Y 446.416,Z 252.498,A -85,B 0,C 180,E1 -8584.523,E2 -8584.523} C_VEL
LIN {X 0,Y 446.425,Z 252.498,A -85,B 0,C 180,E1 -8588.084,E2 -8588.084} C_VEL
LIN {X 0,Y 446.434,Z 252.498,A -85,B 0,C 180,E1 -8590.921,E2 -8590.921} C_VEL
LIN {X 0,Y 446.432,Z 252.498,A -85,B 0,C 180,E1 -8593.841,E2 -8593.841} C_VEL
LIN {X 0,Y 446.433,Z 252.496,A -85,B 0,C 180,E1 -8596.398,E2 -8596.398} C_VEL
LIN {X 0,Y 446.456,Z 252.495,A -85,B 0,C 180,E1 -8599.806,E2 -8599.806} C_VEL
LIN {X 0,Y 446.421,Z 252.497,A -85,B 0,C 180,E1 -8602.125,E2 -8602.125} C_VEL
LIN {X 0,Y 446.418,Z 252.501,A -85,B 0,C 180,E1 -8605.478,E2 -8605.478} C_VEL
LIN {X 0,Y 446.407,Z 252.502,A -85,B 0,C 180,E1 -8608.701,E2 -8608.701} C_VEL
LIN {X 0,Y 446.472,Z 252.491,A -85,B 0,C 180,E1 -8611.822,E2 -8611.822} C_VEL
LIN {X 0,Y 446.447,Z 252.501,A -85,B 0,C 180,E1 -8614.849,E2 -8614.849} C_VEL
LIN {X 0,Y 446.437,Z 252.497,A -85,B 0,C 180,E1 -8618.246,E2 -8618.246} C_VEL
LIN {X 0,Y 446.446,Z 252.495,A -85,B 0,C 180,E1 -8621.65,E2 -8621.65} C_VEL
LIN {X 0,Y 446.497,Z 252.492,A -85,B 0,C 180,E1 -8624.481,E2 -8624.481} C_VEL
LIN {X 0,Y 446.506,Z 252.488,A -85,B 0,C 180,E1 -8627.385,E2 -8627.385} C_VEL
LIN {X 0,Y 446.529,Z 252.488,A -85,B 0,C 180,E1 -8630.946,E2 -8630.946} C_VEL
LIN {X 0,Y 446.639,Z 252.47,A -85,B 0,C 180,E1 -8633.678,E2 -8633.678} C_VEL
LIN {X 0,Y 446.702,Z 252.463,A -85,B 0,C 180,E1 -8637.296,E2 -8637.296} C_VEL
LIN {X 0,Y 446.785,Z 252.454,A -85,B 0,C 180,E1 -8640.001,E2 -8640.001} C_VEL
LIN {X 0,Y 446.702,Z 252.467,A -85,B 0,C 180,E1 -8642.706,E2 -8642.706} C_VEL
LIN {X 0,Y 446.639,Z 252.478,A -85,B 0,C 180,E1 -8646.325,E2 -8646.325} C_VEL
LIN {X 0,Y 446.531,Z 252.484,A -85,B 0,C 180,E1 -8649.057,E2 -8649.057} C_VEL
LIN {X 0,Y 446.516,Z 252.488,A -85,B 0,C 180,E1 -8652.731,E2 -8652.731} C_VEL
LIN {X 0,Y 446.514,Z 252.493,A -85,B 0,C 180,E1 -8656.239,E2 -8656.239} C_VEL
LIN {X 0,Y 446.464,Z 252.492,A -85,B 0,C 180,E1 -8659.304,E2 -8659.304} C_VEL
LIN {X 0,Y 446.414,Z 252.505,A -85,B 0,C 180,E1 -8662.201,E2 -8662.201} C_VEL
LIN {X 0,Y 446.453,Z 252.493,A -85,B 0,C 180,E1 -8665.154,E2 -8665.154} C_VEL
LIN {X 0,Y 446.481,Z 252.495,A -85,B 0,C 180,E1 -8668.18,E2 -8668.18} C_VEL
LIN {X 0,Y 446.417,Z 252.499,A -85,B 0,C 180,E1 -8671.301,E2 -8671.301} C_VEL
LIN {X 0,Y 446.428,Z 252.497,A -85,B 0,C 180,E1 -8674.524,E2 -8674.524} C_VEL
LIN {X 0,Y 446.429,Z 252.501,A -85,B 0,C 180,E1 -8678.083,E2 -8678.083} C_VEL
LIN {X 0,Y 446.425,Z 252.497,A -85,B 0,C 180,E1 -8680.919,E2 -8680.919} C_VEL
LIN {X 0,Y 446.401,Z 252.506,A -85,B 0,C 180,E1 -8683.847,E2 -8683.847} C_VEL
LIN {X 0,Y 446.399,Z 252.501,A -85,B 0,C 180,E1 -8686.404,E2 -8686.404} C_VEL
LIN {X 0,Y 446.426,Z 252.499,A -85,B 0,C 180,E1 -8689.083,E2 -8689.083} C_VEL
LIN {X 0,Y 446.407,Z 252.501,A -85,B 0,C 180,E1 -8692.122,E2 -8692.122} C_VEL
LIN {X 0,Y 446.43,Z 252.504,A -85,B 0,C 180,E1 -8695.478,E2 -8695.478} C_VEL
LIN {X 0,Y 446.417,Z 252.506,A -85,B 0,C 180,E1 -8698.7,E2 -8698.7} C_VEL
LIN {X 0,Y 446.511,Z 252.563,A -85,B 0,C 180,E1 -8701.523,E2 -8701.523} C_VEL
LIN {X 0,Y 450.028,Z 269.191,A -85,B 0,C 180,E1 -8704.617,E2 -8704.617} C_VEL
LIN {X 0,Y 449.205,Z 284.899,A -85,B 0,C 180,E1 -8707.259,E2 -8707.259} C_VEL
LIN {X 0,Y 448.743,Z 292.517,A -85,B 0,C 180,E1 -8708.526,E2 -8708.526} C_VEL
LIN {X 0,Y 453.044,Z 317.136,A -85,B 0,C 180,E1 -8709.136,E2 -8709.136} C_VEL
LIN {X 0,Y 451.76,Z 429.959,A -85,B 0,C 180,E1 -8710.961,E2 -8710.961} C_VEL
LIN {X 0,Y 451.281,Z 444.139,A -85,B 0,C 180,E1 -8711.353,E2 -8711.353} C_VEL
LIN {X 0,Y 450.661,Z 458.732,A -85,B 0,C 180,E1 -8711.958,E2 -8711.958} C_VEL
LIN {X 0,Y 449.933,Z 472.584,A -85,B 0,C 180,E1 -8712.736,E2 -8712.736} C_VEL
LIN {X 0,Y 449.148,Z 485.189,A -85,B 0,C 180,E1 -8713.641,E2 -8713.641} C_VEL
LIN {X 0,Y 448.293,Z 497.875,A -85,B 0,C 180,E1 -8714.776,E2 -8714.776} C_VEL
LIN {X 0,Y 447.551,Z 508.232,A -85,B 0,C 180,E1 -8715.913,E2 -8715.913} C_VEL
LIN {X 0,Y 447.012,Z 518.519,A -85,B 0,C 180,E1 -8717.285,E2 -8717.285} C_VEL
LIN {X 0,Y 446.452,Z 527.031,A -85,B 0,C 180,E1 -8718.652,E2 -8718.652} C_VEL
LIN {X 0,Y 445.966,Z 535.153,A -85,B 0,C 180,E1 -8720.247,E2 -8720.247} C_VEL
LIN {X 0,Y 445.661,Z 541.696,A -85,B 0,C 180,E1 -8721.841,E2 -8721.841} C_VEL
LIN {X 0,Y 445.541,Z 546.235,A -85,B 0,C 180,E1 -8723.206,E2 -8723.206} C_VEL
LIN {X 0,Y 445.461,Z 549.789,A -85,B 0,C 180,E1 -8724.568,E2 -8724.568} C_VEL
LIN {X 0,Y 445.348,Z 553.261,A -85,B 0,C 180,E1 -8726.381,E2 -8726.381} C_VEL
LIN {X 0,Y 445.425,Z 554.469,A -85,B 0,C 180,E1 -8727.287,E2 -8727.287} C_VEL
LIN {X 0,Y 445.337,Z 555.855,A -85,B 0,C 180,E1 -8729.096,E2 -8729.096} C_VEL
LIN {X 0,Y 445.337,Z 555.9,A -85,B 0,C 180,E1 -8730.904,E2 -8730.904} C_VEL
LIN {X 0,Y 445.425,Z 554.605,A -85,B 0,C 180,E1 -8732.713,E2 -8732.713} C_VEL
LIN {X 0,Y 445.394,Z 551.935,A -85,B 0,C 180,E1 -8734.525,E2 -8734.525} C_VEL
LIN {X 0,Y 445.512,Z 547.828,A -85,B 0,C 180,E1 -8736.34,E2 -8736.34} C_VEL
LIN {X 0,Y 445.687,Z 542.165,A -85,B 0,C 180,E1 -8738.159,E2 -8738.159} C_VEL
LIN {X 0,Y 446.006,Z 535.79,A -85,B 0,C 180,E1 -8739.752,E2 -8739.752} C_VEL
LIN {X 0,Y 446.501,Z 527.878,A -85,B 0,C 180,E1 -8741.347,E2 -8741.347} C_VEL
LIN {X 0,Y 447.009,Z 519.631,A -85,B 0,C 180,E1 -8742.715,E2 -8742.715} C_VEL
LIN {X 0,Y 447.718,Z 509.717,A -85,B 0,C 180,E1 -8744.082,E2 -8744.082} C_VEL
LIN {X 0,Y 448.511,Z 498.716,A -85,B 0,C 180,E1 -8745.332,E2 -8745.332} C_VEL
LIN {X 0,Y 449.479,Z 486.482,A -85,B 0,C 180,E1 -8746.463,E2 -8746.463} C_VEL
LIN {X 0,Y 450.292,Z 473.681,A -85,B 0,C 180,E1 -8747.414,E2 -8747.414} C_VEL
LIN {X 0,Y 451.13,Z 459.867,A -85,B 0,C 180,E1 -8748.212,E2 -8748.212} C_VEL
LIN {X 0,Y 451.785,Z 446.289,A -85,B 0,C 180,E1 -8748.802,E2 -8748.802} C_VEL
LIN {X 0,Y 452.291,Z 432.412,A -85,B 0,C 180,E1 -8749.221,E2 -8749.221} C_VEL
LIN {X 0,Y 452.782,Z 406.726,A -85,B 0,C 180,E1 -8749.671,E2 -8749.671} C_VEL
LIN {X 0,Y 453.721,Z 316.689,A -85,B 0,C 180,E1 -8751.144,E2 -8751.144} C_VEL
LIN {X 0,Y 449.931,Z 296.143,A -85,B 0,C 180,E1 -8751.703,E2 -8751.703} C_VEL
LIN {X 0,Y 449.127,Z 292.211,A -85,B 0,C 180,E1 -8751.835,E2 -8751.835} C_VEL
LIN {X 0,Y 450.404,Z 274.241,A -85,B 0,C 180,E1 -8754.916,E2 -8754.916} C_VEL
LIN {X 0,Y 450.39,Z 269.913,A -85,B 0,C 180,E1 -8755.689,E2 -8755.689} C_VEL
LIN {X 0,Y 448.036,Z 259.058,A -85,B 0,C 180,E1 -8757.817,E2 -8757.817} C_VEL
LIN {X 0,Y 446.495,Z 252.492,A -85,B 0,C 180,E1 -8759.175,E2 -8759.175} C_VEL
LIN {X 0,Y 446.423,Z 252.503,A -85,B 0,C 180,E1 -8762.361,E2 -8762.361} C_VEL
LIN {X 0,Y 446.419,Z 252.506,A -85,B 0,C 180,E1 -8765.625,E2 -8765.625} C_VEL
LIN {X 0,Y 446.443,Z 252.502,A -85,B 0,C 180,E1 -8769.026,E2 -8769.026} C_VEL
LIN {X 0,Y 446.45,Z 252.501,A -85,B 0,C 180,E1 -8772.279,E2 -8772.279} C_VEL
LIN {X 0,Y 446.453,Z 252.495,A -85,B 0,C 180,E1 -8775.102,E2 -8775.102} C_VEL
LIN {X 0,Y 446.425,Z 252.502,A -85,B 0,C 180,E1 -8778.608,E2 -8778.608} C_VEL
LIN {X 0,Y 446.441,Z 252.497,A -85,B 0,C 180,E1 -8780.972,E2 -8780.972} C_VEL
LIN {X 0,Y 446.417,Z 252.489,A -85,B 0,C 180,E1 -8784.373,E2 -8784.373} C_VEL
LIN {X 0,Y 446.419,Z 252.502,A -85,B 0,C 180,E1 -8787.637,E2 -8787.637} C_VEL
LIN {X 0,Y 446.464,Z 252.493,A -85,B 0,C 180,E1 -8790.791,E2 -8790.791} C_VEL
LIN {X 0,Y 446.473,Z 252.498,A -85,B 0,C 180,E1 -8793.847,E2 -8793.847} C_VEL
LIN {X 0,Y 446.423,Z 252.497,A -85,B 0,C 180,E1 -8796.822,E2 -8796.822} C_VEL
LIN {X 0,Y 446.437,Z 252.497,A -85,B 0,C 180,E1 -8799.736,E2 -8799.736} C_VEL
LIN {X 0,Y 446.457,Z 252.494,A -85,B 0,C 180,E1 -8802.596,E2 -8802.596} C_VEL
LIN {X 0,Y 446.463,Z 252.496,A -85,B 0,C 180,E1 -8805.411,E2 -8805.411} C_VEL
LIN {X 0,Y 446.511,Z 252.483,A -85,B 0,C 180,E1 -8808.192,E2 -8808.192} C_VEL
LIN {X 0,Y 446.592,Z 252.475,A -85,B 0,C 180,E1 -8811.857,E2 -8811.857} C_VEL
LIN {X 0,Y 446.637,Z 252.472,A -85,B 0,C 180,E1 -8814.581,E2 -8814.581} C_VEL
LIN {X 0,Y 446.7,Z 252.464,A -85,B 0,C 180,E1 -8817.293,E2 -8817.293} C_VEL
LIN {X 0,Y 446.784,Z 252.453,A -85,B 0,C 180,E1 -8819.999,E2 -8819.999} C_VEL
LIN {X 0,Y 446.7,Z 252.464,A -85,B 0,C 180,E1 -8822.704,E2 -8822.704} C_VEL
LIN {X 0,Y 446.636,Z 252.469,A -85,B 0,C 180,E1 -8826.323,E2 -8826.323} C_VEL
LIN {X 0,Y 446.528,Z 252.487,A -85,B 0,C 180,E1 -8829.054,E2 -8829.054} C_VEL
LIN {X 0,Y 446.51,Z 252.492,A -85,B 0,C 180,E1 -8832.729,E2 -8832.729} C_VEL
LIN {X 0,Y 446.484,Z 252.492,A -85,B 0,C 180,E1 -8836.227,E2 -8836.227} C_VEL
LIN {X 0,Y 446.458,Z 252.496,A -85,B 0,C 180,E1 -8839.302,E2 -8839.302} C_VEL
LIN {X 0,Y 446.42,Z 252.5,A -85,B 0,C 180,E1 -8842.198,E2 -8842.198} C_VEL
LIN {X 0,Y 446.445,Z 252.499,A -85,B 0,C 180,E1 -8845.151,E2 -8845.151} C_VEL
LIN {X 0,Y 446.471,Z 252.495,A -85,B 0,C 180,E1 -8848.178,E2 -8848.178} C_VEL
LIN {X 0,Y 446.405,Z 252.497,A -85,B 0,C 180,E1 -8851.299,E2 -8851.299} C_VEL
LIN {X 0,Y 446.416,Z 252.497,A -85,B 0,C 180,E1 -8854.522,E2 -8854.522} C_VEL
LIN {X 0,Y 446.423,Z 252.503,A -85,B 0,C 180,E1 -8858.082,E2 -8858.082} C_VEL
LIN {X 0,Y 446.433,Z 252.5,A -85,B 0,C 180,E1 -8860.92,E2 -8860.92} C_VEL
LIN {X 0,Y 446.43,Z 252.502,A -85,B 0,C 180,E1 -8863.84,E2 -8863.84} C_VEL
LIN {X 0,Y 446.432,Z 252.503,A -85,B 0,C 180,E1 -8866.396,E2 -8866.396} C_VEL
LIN {X 0,Y 446.456,Z 252.502,A -85,B 0,C 180,E1 -8869.805,E2 -8869.805} C_VEL
LIN {X 0,Y 446.501,Z 252.66,A -85,B 0,C 180,E1 -8870.465,E2 -8870.465} C_VEL
LIN {X 0,Y 449.051,Z 264.63,A -85,B 0,C 180,E1 -8873.129,E2 -8873.129} C_VEL
LIN {X 0,Y 449.546,Z 268.977,A -85,B 0,C 180,E1 -8874.047,E2 -8874.047} C_VEL
LIN {X 0,Y 449.466,Z 270.02,A -85,B 0,C 180,E1 -8874.253,E2 -8874.253} C_VEL
LIN {X 0,Y 453.864,Z 289.061,A -85,B 0,C 180,E1 -8874.829,E2 -8874.829} C_VEL
LIN {X 0,Y 454.137,Z 293.313,A -85,B 0,C 180,E1 -8874.917,E2 -8874.917} C_VEL
LIN {X 0,Y 452.592,Z 406.939,A -85,B 0,C 180,E1 -8876.786,E2 -8876.786} C_VEL
LIN {X 0,Y 452.163,Z 421.356,A -85,B 0,C 180,E1 -8877.21,E2 -8877.21} C_VEL
LIN {X 0,Y 451.538,Z 434.91,A -85,B 0,C 180,E1 -8877.787,E2 -8877.787} C_VEL
LIN {X 0,Y 450.875,Z 447.839,A -85,B 0,C 180,E1 -8878.522,E2 -8878.522} C_VEL
LIN {X 0,Y 450.032,Z 460.547,A -85,B 0,C 180,E1 -8879.44,E2 -8879.44} C_VEL
LIN {X 0,Y 449.215,Z 472.076,A -85,B 0,C 180,E1 -8880.475,E2 -8880.475} C_VEL
LIN {X 0,Y 448.426,Z 482.325,A -85,B 0,C 180,E1 -8881.589,E2 -8881.589} C_VEL
LIN {X 0,Y 448.235,Z 484.609,A -85,B 0,C 180,E1 -8881.863,E2 -8881.863} C_VEL
LIN {X 0,Y 447.236,Z 488.865,A -85,B 0,C 180,E1 -8882.384,E2 -8882.384} C_VEL
LIN {X 0,Y 443.929,Z 495.474,A -85,B 0,C 180,E1 -8883.236,E2 -8883.236} C_VEL
LIN {X 0,Y 440.697,Z 501.63,A -85,B 0,C 180,E1 -8884.15,E2 -8884.15} C_VEL
LIN {X 0,Y 439.817,Z 505.027,A -85,B 0,C 180,E1 -8884.76,E2 -8884.76} C_VEL
LIN {X 0,Y 439.239,Z 512.75,A -85,B 0,C 180,E1 -8886.422,E2 -8886.422} C_VEL
LIN {X 0,Y 438.876,Z 518.229,A -85,B 0,C 180,E1 -8887.89,E2 -8887.89} C_VEL
LIN {X 0,Y 438.591,Z 522.652,A -85,B 0,C 180,E1 -8889.359,E2 -8889.359} C_VEL
LIN {X 0,Y 438.419,Z 526.521,A -85,B 0,C 180,E1 -8891.042,E2 -8891.042} C_VEL
LIN {X 0,Y 438.247,Z 528.597,A -85,B 0,C 180,E1 -8892.261,E2 -8892.261} C_VEL
LIN {X 0,Y 438.229,Z 530.647,A -85,B 0,C 180,E1 -8894.197,E2 -8894.197} C_VEL
LIN {X 0,Y 438.154,Z 531.217,A -85,B 0,C 180,E1 -8896.078,E2 -8896.078} C_VEL
LIN {X 0,Y 438.255,Z 530.366,A -85,B 0,C 180,E1 -8898.009,E2 -8898.009} C_VEL
LIN {X 0,Y 438.265,Z 528.219,A -85,B 0,C 180,E1 -8899.84,E2 -8899.84} C_VEL
LIN {X 0,Y 438.469,Z 524.617,A -85,B 0,C 180,E1 -8901.706,E2 -8901.706} C_VEL
LIN {X 0,Y 438.688,Z 519.523,A -85,B 0,C 180,E1 -8903.561,E2 -8903.561} C_VEL
LIN {X 0,Y 438.905,Z 514.598,A -85,B 0,C 180,E1 -8904.948,E2 -8904.948} C_VEL
LIN {X 0,Y 439.357,Z 507.537,A -85,B 0,C 180,E1 -8906.561,E2 -8906.561} C_VEL
LIN {X 0,Y 439.958,Z 498.828,A -85,B 0,C 180,E1 -8908.169,E2 -8908.169} C_VEL
LIN {X 0,Y 440.623,Z 489.729,A -85,B 0,C 180,E1 -8909.543,E2 -8909.543} C_VEL
LIN {X 0,Y 441.448,Z 478.701,A -85,B 0,C 180,E1 -8910.912,E2 -8910.912} C_VEL
LIN {X 0,Y 442.295,Z 467.46,A -85,B 0,C 180,E1 -8912.049,E2 -8912.049} C_VEL
LIN {X 0,Y 443.093,Z 455.078,A -85,B 0,C 180,E1 -8913.069,E2 -8913.069} C_VEL
LIN {X 0,Y 443.824,Z 441.612,A -85,B 0,C 180,E1 -8913.949,E2 -8913.949} C_VEL
LIN {X 0,Y 444.409,Z 428.507,A -85,B 0,C 180,E1 -8914.606,E2 -8914.606} C_VEL
LIN {X 0,Y 444.911,Z 414.177,A -85,B 0,C 180,E1 -8915.126,E2 -8915.126} C_VEL
LIN {X 0,Y 445.213,Z 399.421,A -85,B 0,C 180,E1 -8915.463,E2 -8915.463} C_VEL
LIN {X 0,Y 446.546,Z 291.875,A -85,B 0,C 180,E1 -8917.209,E2 -8917.209} C_VEL
LIN {X 0,Y 442.711,Z 273.448,A -85,B 0,C 180,E1 -8917.695,E2 -8917.695} C_VEL
LIN {X 0,Y 442.012,Z 269.817,A -85,B 0,C 180,E1 -8917.816,E2 -8917.816} C_VEL
LIN {X 0,Y 441.925,Z 265.46,A -85,B 0,C 180,E1 -8918.689,E2 -8918.689} C_VEL
LIN {X 0,Y 439.517,Z 253.365,A -85,B 0,C 180,E1 -8921.296,E2 -8921.296} C_VEL
LIN {X 0,Y 439.424,Z 253.377,A -85,B 0,C 180,E1 -8923.881,E2 -8923.881} C_VEL
LIN {X 0,Y 439.436,Z 253.368,A -85,B 0,C 180,E1 -8926.731,E2 -8926.731} C_VEL
LIN {X 0,Y 439.417,Z 253.376,A -85,B 0,C 180,E1 -8929.625,E2 -8929.625} C_VEL
LIN {X 0,Y 439.351,Z 253.378,A -85,B 0,C 180,E1 -8932.576,E2 -8932.576} C_VEL
LIN {X 0,Y 439.4,Z 253.379,A -85,B 0,C 180,E1 -8935.585,E2 -8935.585} C_VEL
LIN {X 0,Y 439.411,Z 253.371,A -85,B 0,C 180,E1 -8938.673,E2 -8938.673} C_VEL
LIN {X 0,Y 439.369,Z 253.378,A -85,B 0,C 180,E1 -8942.034,E2 -8942.034} C_VEL
LIN {X 0,Y 439.382,Z 253.38,A -85,B 0,C 180,E1 -8945.341,E2 -8945.341} C_VEL
LIN {X 0,Y 439.387,Z 253.374,A -85,B 0,C 180,E1 -8948.594,E2 -8948.594} C_VEL
LIN {X 0,Y 439.392,Z 253.379,A -85,B 0,C 180,E1 -8951.26,E2 -8951.26} C_VEL
LIN {X 0,Y 439.396,Z 253.374,A -85,B 0,C 180,E1 -8954.729,E2 -8954.729} C_VEL
LIN {X 0,Y 439.399,Z 253.374,A -85,B 0,C 180,E1 -8957.798,E2 -8957.798} C_VEL
LIN {X 0,Y 439.439,Z 253.367,A -85,B 0,C 180,E1 -8960.231,E2 -8960.231} C_VEL
LIN {X 0,Y 439.365,Z 253.378,A -85,B 0,C 180,E1 -8963.714,E2 -8963.714} C_VEL
LIN {X 0,Y 439.361,Z 253.384,A -85,B 0,C 180,E1 -8967.055,E2 -8967.055} C_VEL
LIN {X 0,Y 439.384,Z 253.374,A -85,B 0,C 180,E1 -8970.276,E2 -8970.276} C_VEL
LIN {X 0,Y 439.422,Z 253.371,A -85,B 0,C 180,E1 -8973.59,E2 -8973.59} C_VEL
LIN {X 0,Y 439.375,Z 253.377,A -85,B 0,C 180,E1 -8976.431,E2 -8976.431} C_VEL
LIN {X 0,Y 439.377,Z 253.377,A -85,B 0,C 180,E1 -8979.398,E2 -8979.398} C_VEL
LIN {X 0,Y 439.421,Z 253.371,A -85,B 0,C 180,E1 -8982.311,E2 -8982.311} C_VEL
LIN {X 0,Y 439.439,Z 253.37,A -85,B 0,C 180,E1 -8985.175,E2 -8985.175} C_VEL
LIN {X 0,Y 439.474,Z 253.364,A -85,B 0,C 180,E1 -8988.002,E2 -8988.002} C_VEL
LIN {X 0,Y 439.539,Z 253.355,A -85,B 0,C 180,E1 -8991.727,E2 -8991.727} C_VEL
LIN {X 0,Y 439.615,Z 253.352,A -85,B 0,C 180,E1 -8994.497,E2 -8994.497} C_VEL
LIN {X 0,Y 439.628,Z 253.347,A -85,B 0,C 180,E1 -8998.169,E2 -8998.169} C_VEL
LIN {X 0,Y 439.755,Z 253.33,A -85,B 0,C 180,E1 -9000.001,E2 -9000.001} C_VEL
LIN {X 0,Y 439.649,Z 253.345,A -85,B 0,C 180,E1 -9002.75,E2 -9002.75} C_VEL
LIN {X 0,Y 439.611,Z 253.353,A -85,B 0,C 180,E1 -9006.426,E2 -9006.426} C_VEL
LIN {X 0,Y 439.493,Z 253.361,A -85,B 0,C 180,E1 -9009.203,E2 -9009.203} C_VEL
LIN {X 0,Y 439.46,Z 253.365,A -85,B 0,C 180,E1 -9012.939,E2 -9012.939} C_VEL
LIN {X 0,Y 439.455,Z 253.371,A -85,B 0,C 180,E1 -9016.356,E2 -9016.356} C_VEL
LIN {X 0,Y 439.398,Z 253.374,A -85,B 0,C 180,E1 -9019.628,E2 -9019.628} C_VEL
LIN {X 0,Y 439.361,Z 253.379,A -85,B 0,C 180,E1 -9022.577,E2 -9022.577} C_VEL
LIN {X 0,Y 439.401,Z 253.374,A -85,B 0,C 180,E1 -9025.586,E2 -9025.586} C_VEL
LIN {X 0,Y 439.422,Z 253.37,A -85,B 0,C 180,E1 -9028.674,E2 -9028.674} C_VEL
LIN {X 0,Y 439.38,Z 253.381,A -85,B 0,C 180,E1 -9032.034,E2 -9032.034} C_VEL
LIN {X 0,Y 439.394,Z 253.375,A -85,B 0,C 180,E1 -9035.342,E2 -9035.342} C_VEL
LIN {X 0,Y 439.388,Z 253.374,A -85,B 0,C 180,E1 -9038.595,E2 -9038.595} C_VEL
LIN {X 0,Y 439.387,Z 253.376,A -85,B 0,C 180,E1 -9041.258,E2 -9041.258} C_VEL
LIN {X 0,Y 439.401,Z 253.372,A -85,B 0,C 180,E1 -9044.73,E2 -9044.73} C_VEL
LIN {X 0,Y 439.396,Z 253.378,A -85,B 0,C 180,E1 -9047.797,E2 -9047.797} C_VEL
LIN {X 0,Y 439.389,Z 253.374,A -85,B 0,C 180,E1 -9050.224,E2 -9050.224} C_VEL
LIN {X 0,Y 439.374,Z 253.38,A -85,B 0,C 180,E1 -9053.714,E2 -9053.714} C_VEL
LIN {X 0,Y 439.374,Z 253.378,A -85,B 0,C 180,E1 -9057.055,E2 -9057.055} C_VEL
LIN {X 0,Y 439.42,Z 253.377,A -85,B 0,C 180,E1 -9060.804,E2 -9060.804} C_VEL
LIN {X 0,Y 439.457,Z 253.425,A -85,B 0,C 180,E1 -9061.265,E2 -9061.265} C_VEL
LIN {X 0,Y 442.675,Z 268.443,A -85,B 0,C 180,E1 -9064.114,E2 -9064.114} C_VEL
LIN {X 0,Y 443.087,Z 272.455,A -85,B 0,C 180,E1 -9064.837,E2 -9064.837} C_VEL
LIN {X 0,Y 441.878,Z 292.107,A -85,B 0,C 180,E1 -9068.176,E2 -9068.176} C_VEL
LIN {X 0,Y 441.891,Z 292.679,A -85,B 0,C 180,E1 -9068.233,E2 -9068.233} C_VEL
LIN {X 0,Y 446.348,Z 318.296,A -85,B 0,C 180,E1 -9068.865,E2 -9068.865} C_VEL
LIN {X 0,Y 444.962,Z 430.897,A -85,B 0,C 180,E1 -9070.719,E2 -9070.719} C_VEL
LIN {X 0,Y 444.44,Z 445.417,A -85,B 0,C 180,E1 -9071.145,E2 -9071.145} C_VEL
LIN {X 0,Y 443.842,Z 458.35,A -85,B 0,C 180,E1 -9071.693,E2 -9071.693} C_VEL
LIN {X 0,Y 443.12,Z 471.908,A -85,B 0,C 180,E1 -9072.462,E2 -9072.462} C_VEL
LIN {X 0,Y 442.285,Z 484.603,A -85,B 0,C 180,E1 -9073.38,E2 -9073.38} C_VEL
LIN {X 0,Y 441.52,Z 496.178,A -85,B 0,C 180,E1 -9074.419,E2 -9074.419} C_VEL
LIN {X 0,Y 440.781,Z 505.805,A -85,B 0,C 180,E1 -9075.456,E2 -9075.456} C_VEL
LIN {X 0,Y 440.063,Z 516.677,A -85,B 0,C 180,E1 -9076.869,E2 -9076.869} C_VEL
LIN {X 0,Y 439.51,Z 525.339,A -85,B 0,C 180,E1 -9078.236,E2 -9078.236} C_VEL
LIN {X 0,Y 438.942,Z 533.796,A -85,B 0,C 180,E1 -9079.856,E2 -9079.856} C_VEL
LIN {X 0,Y 438.678,Z 539.683,A -85,B 0,C 180,E1 -9081.246,E2 -9081.246} C_VEL
LIN {X 0,Y 438.459,Z 545.968,A -85,B 0,C 180,E1 -9083.095,E2 -9083.095} C_VEL
LIN {X 0,Y 438.359,Z 549.536,A -85,B 0,C 180,E1 -9084.48,E2 -9084.48} C_VEL
LIN {X 0,Y 438.252,Z 553.026,A -85,B 0,C 180,E1 -9086.322,E2 -9086.322} C_VEL
LIN {X 0,Y 438.332,Z 554.242,A -85,B 0,C 180,E1 -9087.243,E2 -9087.243} C_VEL
LIN {X 0,Y 438.251,Z 555.643,A -85,B 0,C 180,E1 -9089.081,E2 -9089.081} C_VEL
LIN {X 0,Y 438.251,Z 555.705,A -85,B 0,C 180,E1 -9090.919,E2 -9090.919} C_VEL
LIN {X 0,Y 438.331,Z 554.428,A -85,B 0,C 180,E1 -9092.757,E2 -9092.757} C_VEL
LIN {X 0,Y 438.319,Z 551.777,A -85,B 0,C 180,E1 -9094.598,E2 -9094.598} C_VEL
LIN {X 0,Y 438.432,Z 547.69,A -85,B 0,C 180,E1 -9096.442,E2 -9096.442} C_VEL
LIN {X 0,Y 438.622,Z 542.052,A -85,B 0,C 180,E1 -9098.291,E2 -9098.291} C_VEL
LIN {X 0,Y 438.939,Z 535.708,A -85,B 0,C 180,E1 -9099.911,E2 -9099.911} C_VEL
LIN {X 0,Y 439.507,Z 527.831,A -85,B 0,C 180,E1 -9101.53,E2 -9101.53} C_VEL
LIN {X 0,Y 440.088,Z 518.745,A -85,B 0,C 180,E1 -9103.056,E2 -9103.056} C_VEL
LIN {X 0,Y 440.785,Z 509.739,A -85,B 0,C 180,E1 -9104.308,E2 -9104.308} C_VEL
LIN {X 0,Y 441.659,Z 498.782,A -85,B 0,C 180,E1 -9105.576,E2 -9105.576} C_VEL
LIN {X 0,Y 442.674,Z 486.628,A -85,B 0,C 180,E1 -9106.723,E2 -9106.723} C_VEL
LIN {X 0,Y 443.521,Z 474.105,A -85,B 0,C 180,E1 -9107.677,E2 -9107.677} C_VEL
LIN {X 0,Y 444.365,Z 461.398,A -85,B 0,C 180,E1 -9108.44,E2 -9108.44} C_VEL
LIN {X 0,Y 445.061,Z 447.694,A -85,B 0,C 180,E1 -9109.067,E2 -9109.067} C_VEL
LIN {X 0,Y 445.63,Z 433.512,A -85,B 0,C 180,E1 -9109.52,E2 -9109.52} C_VEL
LIN {X 0,Y 446.068,Z 413.904,A -85,B 0,C 180,E1 -9109.89,E2 -9109.89} C_VEL
LIN {X 0,Y 447.227,Z 317.752,A -85,B 0,C 180,E1 -9111.482,E2 -9111.482} C_VEL
LIN {X 0,Y 443.276,Z 296.554,A -85,B 0,C 180,E1 -9112.076,E2 -9112.076} C_VEL
LIN {X 0,Y 442.344,Z 292.06,A -85,B 0,C 180,E1 -9112.221,E2 -9112.221} C_VEL
LIN {X 0,Y 443.719,Z 273.487,A -85,B 0,C 180,E1 -9115.468,E2 -9115.468} C_VEL
LIN {X 0,Y 442.425,Z 266.011,A -85,B 0,C 180,E1 -9116.923,E2 -9116.923} C_VEL
LIN {X 0,Y 439.43,Z 253.374,A -85,B 0,C 180,E1 -9119.524,E2 -9119.524} C_VEL
LIN {X 0,Y 439.373,Z 253.384,A -85,B 0,C 180,E1 -9122.945,E2 -9122.945} C_VEL
LIN {X 0,Y 439.373,Z 253.388,A -85,B 0,C 180,E1 -9126.286,E2 -9126.286} C_VEL
LIN {X 0,Y 439.401,Z 253.38,A -85,B 0,C 180,E1 -9129.848,E2 -9129.848} C_VEL
LIN {X 0,Y 439.402,Z 253.378,A -85,B 0,C 180,E1 -9132.629,E2 -9132.629} C_VEL
LIN {X 0,Y 439.401,Z 253.374,A -85,B 0,C 180,E1 -9135.27,E2 -9135.27} C_VEL
LIN {X 0,Y 439.386,Z 253.377,A -85,B 0,C 180,E1 -9138.742,E2 -9138.742} C_VEL
LIN {X 0,Y 439.371,Z 253.379,A -85,B 0,C 180,E1 -9141.606,E2 -9141.606} C_VEL
LIN {X 0,Y 439.397,Z 253.364,A -85,B 0,C 180,E1 -9144.843,E2 -9144.843} C_VEL
LIN {X 0,Y 439.37,Z 253.378,A -85,B 0,C 180,E1 -9148.138,E2 -9148.138} C_VEL
LIN {X 0,Y 439.42,Z 253.372,A -85,B 0,C 180,E1 -9151.326,E2 -9151.326} C_VEL
LIN {X 0,Y 439.4,Z 253.374,A -85,B 0,C 180,E1 -9154.414,E2 -9154.414} C_VEL
LIN {X 0,Y 439.359,Z 253.38,A -85,B 0,C 180,E1 -9157.423,E2 -9157.423} C_VEL
LIN {X 0,Y 439.435,Z 253.367,A -85,B 0,C 180,E1 -9160.662,E2 -9160.662} C_VEL
LIN {X 0,Y 439.455,Z 253.365,A -85,B 0,C 180,E1 -9164.223,E2 -9164.223} C_VEL
LIN {X 0,Y 439.477,Z 253.361,A -85,B 0,C 180,E1 -9168,E2 -9168} C_VEL
LIN {X 0,Y 439.54,Z 253.354,A -85,B 0,C 180,E1 -9171.725,E2 -9171.725} C_VEL
LIN {X 0,Y 439.613,Z 253.347,A -85,B 0,C 180,E1 -9174.495,E2 -9174.495} C_VEL
LIN {X 0,Y 439.627,Z 253.344,A -85,B 0,C 180,E1 -9178.167,E2 -9178.167} C_VEL
LIN {X 0,Y 439.755,Z 253.328,A -85,B 0,C 180,E1 -9179.999,E2 -9179.999} C_VEL
LIN {X 0,Y 439.647,Z 253.342,A -85,B 0,C 180,E1 -9182.747,E2 -9182.747} C_VEL
LIN {X 0,Y 439.607,Z 253.345,A -85,B 0,C 180,E1 -9186.424,E2 -9186.424} C_VEL
LIN {X 0,Y 439.489,Z 253.362,A -85,B 0,C 180,E1 -9189.2,E2 -9189.2} C_VEL
LIN {X 0,Y 439.454,Z 253.369,A -85,B 0,C 180,E1 -9192.937,E2 -9192.937} C_VEL
LIN {X 0,Y 439.435,Z 253.37,A -85,B 0,C 180,E1 -9196.348,E2 -9196.348} C_VEL
LIN {X 0,Y 439.422,Z 253.37,A -85,B 0,C 180,E1 -9199.624,E2 -9199.624} C_VEL
LIN {X 0,Y 439.361,Z 253.383,A -85,B 0,C 180,E1 -9202.574,E2 -9202.574} C_VEL
LIN {X 0,Y 439.392,Z 253.375,A -85,B 0,C 180,E1 -9205.584,E2 -9205.584} C_VEL
LIN {X 0,Y 439.411,Z 253.377,A -85,B 0,C 180,E1 -9208.672,E2 -9208.672} C_VEL
LIN {X 0,Y 439.36,Z 253.374,A -85,B 0,C 180,E1 -9211.86,E2 -9211.86} C_VEL
LIN {X 0,Y 439.386,Z 253.369,A -85,B 0,C 180,E1 -9215.155,E2 -9215.155} C_VEL
LIN {X 0,Y 439.383,Z 253.374,A -85,B 0,C 180,E1 -9218.593,E2 -9218.593} C_VEL
LIN {X 0,Y 439.39,Z 253.376,A -85,B 0,C 180,E1 -9221.259,E2 -9221.259} C_VEL
LIN {X 0,Y 439.395,Z 253.378,A -85,B 0,C 180,E1 -9224.728,E2 -9224.728} C_VEL
LIN {X 0,Y 439.398,Z 253.378,A -85,B 0,C 180,E1 -9227.797,E2 -9227.797} C_VEL
LIN {X 0,Y 439.461,Z 253.466,A -85,B 0,C 180,E1 -9230.101,E2 -9230.101} C_VEL
LIN {X 0,Y 442.328,Z 266.984,A -85,B 0,C 180,E1 -9233.161,E2 -9233.161} C_VEL
LIN {X 0,Y 442.74,Z 270.355,A -85,B 0,C 180,E1 -9233.866,E2 -9233.866} C_VEL
LIN {X 0,Y 446.898,Z 288.008,A -85,B 0,C 180,E1 -9234.419,E2 -9234.419} C_VEL
LIN {X 0,Y 447.646,Z 292.334,A -85,B 0,C 180,E1 -9234.537,E2 -9234.537} C_VEL
LIN {X 0,Y 446.045,Z 406.171,A -85,B 0,C 180,E1 -9236.432,E2 -9236.432} C_VEL
LIN {X 0,Y 445.589,Z 420.382,A -85,B 0,C 180,E1 -9236.839,E2 -9236.839} C_VEL
LIN {X 0,Y 444.957,Z 433.819,A -85,B 0,C 180,E1 -9237.403,E2 -9237.403} C_VEL
LIN {X 0,Y 444.225,Z 446.748,A -85,B 0,C 180,E1 -9238.129,E2 -9238.129} C_VEL
LIN {X 0,Y 443.423,Z 459.314,A -85,B 0,C 180,E1 -9239.033,E2 -9239.033} C_VEL
LIN {X 0,Y 442.45,Z 471.387,A -85,B 0,C 180,E1 -9240.109,E2 -9240.109} C_VEL
LIN {X 0,Y 441.599,Z 482.377,A -85,B 0,C 180,E1 -9241.312,E2 -9241.312} C_VEL
LIN {X 0,Y 440.767,Z 492.862,A -85,B 0,C 180,E1 -9242.708,E2 -9242.708} C_VEL
LIN {X 0,Y 440.062,Z 502.067,A -85,B 0,C 180,E1 -9244.203,E2 -9244.203} C_VEL
LIN {X 0,Y 439.817,Z 505.027,A -85,B 0,C 180,E1 -9244.76,E2 -9244.76} C_VEL
LIN {X 0,Y 438.945,Z 508.303,A -85,B 0,C 180,E1 -9245.392,E2 -9245.392} C_VEL
LIN {X 0,Y 435.764,Z 513.318,A -85,B 0,C 180,E1 -9246.433,E2 -9246.433} C_VEL
LIN {X 0,Y 432.587,Z 517.736,A -85,B 0,C 180,E1 -9247.53,E2 -9247.53} C_VEL
LIN {X 0,Y 431.74,Z 520.079,A -85,B 0,C 180,E1 -9248.242,E2 -9248.242} C_VEL
LIN {X 0,Y 431.448,Z 524.771,A -85,B 0,C 180,E1 -9249.997,E2 -9249.997} C_VEL
LIN {X 0,Y 431.215,Z 528.481,A -85,B 0,C 180,E1 -9251.962,E2 -9251.962} C_VEL
LIN {X 0,Y 431.112,Z 530.671,A -85,B 0,C 180,E1 -9253.911,E2 -9253.911} C_VEL
LIN {X 0,Y 431.057,Z 531.428,A -85,B 0,C 180,E1 -9255.845,E2 -9255.845} C_VEL
LIN {X 0,Y 431.141,Z 530.775,A -85,B 0,C 180,E1 -9257.766,E2 -9257.766} C_VEL
LIN {X 0,Y 431.161,Z 528.729,A -85,B 0,C 180,E1 -9259.671,E2 -9259.671} C_VEL
LIN {X 0,Y 431.355,Z 525.27,A -85,B 0,C 180,E1 -9261.568,E2 -9261.568} C_VEL
LIN {X 0,Y 431.594,Z 520.323,A -85,B 0,C 180,E1 -9263.455,E2 -9263.455} C_VEL
LIN {X 0,Y 431.958,Z 513.748,A -85,B 0,C 180,E1 -9265.334,E2 -9265.334} C_VEL
LIN {X 0,Y 432.398,Z 506.456,A -85,B 0,C 180,E1 -9266.972,E2 -9266.972} C_VEL
LIN {X 0,Y 433.087,Z 497.402,A -85,B 0,C 180,E1 -9268.605,E2 -9268.605} C_VEL
LIN {X 0,Y 433.845,Z 487.947,A -85,B 0,C 180,E1 -9270,E2 -9270} C_VEL
LIN {X 0,Y 434.617,Z 477.512,A -85,B 0,C 180,E1 -9271.274,E2 -9271.274} C_VEL
LIN {X 0,Y 435.51,Z 465.972,A -85,B 0,C 180,E1 -9272.428,E2 -9272.428} C_VEL
LIN {X 0,Y 436.376,Z 453.19,A -85,B 0,C 180,E1 -9273.463,E2 -9273.463} C_VEL
LIN {X 0,Y 437.073,Z 440.724,A -85,B 0,C 180,E1 -9274.265,E2 -9274.265} C_VEL
LIN {X 0,Y 437.727,Z 427.138,A -85,B 0,C 180,E1 -9274.936,E2 -9274.936} C_VEL
LIN {X 0,Y 438.165,Z 413.235,A -85,B 0,C 180,E1 -9275.431,E2 -9275.431} C_VEL
LIN {X 0,Y 438.44,Z 398.892,A -85,B 0,C 180,E1 -9275.75,E2 -9275.75} C_VEL
LIN {X 0,Y 439.784,Z 291.821,A -85,B 0,C 180,E1 -9277.516,E2 -9277.516} C_VEL
LIN {X 0,Y 435.146,Z 270.022,A -85,B 0,C 180,E1 -9278.133,E2 -9278.133} C_VEL
LIN {X 0,Y 434.957,Z 266.616,A -85,B 0,C 180,E1 -9278.83,E2 -9278.83} C_VEL
LIN {X 0,Y 432.449,Z 254.246,A -85,B 0,C 180,E1 -9281.543,E2 -9281.543} C_VEL
LIN {X 0,Y 432.371,Z 254.26,A -85,B 0,C 180,E1 -9284.112,E2 -9284.112} C_VEL
LIN {X 0,Y 432.383,Z 254.246,A -85,B 0,C 180,E1 -9287.012,E2 -9287.012} C_VEL
LIN {X 0,Y 432.359,Z 254.254,A -85,B 0,C 180,E1 -9289.959,E2 -9289.959} C_VEL
LIN {X 0,Y 432.306,Z 254.256,A -85,B 0,C 180,E1 -9292.965,E2 -9292.965} C_VEL
LIN {X 0,Y 432.354,Z 254.253,A -85,B 0,C 180,E1 -9296.033,E2 -9296.033} C_VEL
LIN {X 0,Y 432.339,Z 254.254,A -85,B 0,C 180,E1 -9299.187,E2 -9299.187} C_VEL
LIN {X 0,Y 432.318,Z 254.255,A -85,B 0,C 180,E1 -9302.295,E2 -9302.295} C_VEL
LIN {X 0,Y 432.327,Z 254.253,A -85,B 0,C 180,E1 -9304.677,E2 -9304.677} C_VEL
LIN {X 0,Y 432.34,Z 254.252,A -85,B 0,C 180,E1 -9308.149,E2 -9308.149} C_VEL
LIN {X 0,Y 432.36,Z 254.254,A -85,B 0,C 180,E1 -9311.609,E2 -9311.609} C_VEL
LIN {X 0,Y 432.365,Z 254.248,A -85,B 0,C 180,E1 -9314.342,E2 -9314.342} C_VEL
LIN {X 0,Y 432.353,Z 254.254,A -85,B 0,C 180,E1 -9317.01,E2 -9317.01} C_VEL
LIN {X 0,Y 432.345,Z 254.252,A -85,B 0,C 180,E1 -9319.818,E2 -9319.818} C_VEL
LIN {X 0,Y 432.305,Z 254.262,A -85,B 0,C 180,E1 -9323.024,E2 -9323.024} C_VEL
LIN {X 0,Y 432.347,Z 254.251,A -85,B 0,C 180,E1 -9325.997,E2 -9325.997} C_VEL
LIN {X 0,Y 432.383,Z 254.247,A -85,B 0,C 180,E1 -9329.745,E2 -9329.745} C_VEL
LIN {X 0,Y 432.388,Z 254.248,A -85,B 0,C 180,E1 -9333.373,E2 -9333.373} C_VEL
LIN {X 0,Y 432.36,Z 254.249,A -85,B 0,C 180,E1 -9336.024,E2 -9336.024} C_VEL
LIN {X 0,Y 432.339,Z 254.257,A -85,B 0,C 180,E1 -9339.047,E2 -9339.047} C_VEL
LIN {X 0,Y 432.367,Z 254.248,A -85,B 0,C 180,E1 -9342.012,E2 -9342.012} C_VEL
LIN {X 0,Y 432.386,Z 254.251,A -85,B 0,C 180,E1 -9344.928,E2 -9344.928} C_VEL
LIN {X 0,Y 432.449,Z 254.238,A -85,B 0,C 180,E1 -9347.805,E2 -9347.805} C_VEL
LIN {X 0,Y 432.483,Z 254.234,A -85,B 0,C 180,E1 -9351.592,E2 -9351.592} C_VEL
LIN {X 0,Y 432.591,Z 254.225,A -85,B 0,C 180,E1 -9354.407,E2 -9354.407} C_VEL
LIN {X 0,Y 432.598,Z 254.222,A -85,B 0,C 180,E1 -9358.139,E2 -9358.139} C_VEL
LIN {X 0,Y 432.725,Z 254.206,A -85,B 0,C 180,E1 -9360.001,E2 -9360.001} C_VEL
LIN {X 0,Y 432.598,Z 254.223,A -85,B 0,C 180,E1 -9362.795,E2 -9362.795} C_VEL
LIN {X 0,Y 432.566,Z 254.229,A -85,B 0,C 180,E1 -9366.532,E2 -9366.532} C_VEL
LIN {X 0,Y 432.437,Z 254.24,A -85,B 0,C 180,E1 -9369.354,E2 -9369.354} C_VEL
LIN {X 0,Y 432.425,Z 254.243,A -85,B 0,C 180,E1 -9372.805,E2 -9372.805} C_VEL
LIN {X 0,Y 432.418,Z 254.246,A -85,B 0,C 180,E1 -9376.485,E2 -9376.485} C_VEL
LIN {X 0,Y 432.334,Z 254.258,A -85,B 0,C 180,E1 -9379.962,E2 -9379.962} C_VEL
LIN {X 0,Y 432.315,Z 254.255,A -85,B 0,C 180,E1 -9382.965,E2 -9382.965} C_VEL
LIN {X 0,Y 432.361,Z 254.257,A -85,B 0,C 180,E1 -9386.034,E2 -9386.034} C_VEL
LIN {X 0,Y 432.349,Z 254.251,A -85,B 0,C 180,E1 -9389.188,E2 -9389.188} C_VEL
LIN {X 0,Y 432.329,Z 254.256,A -85,B 0,C 180,E1 -9392.296,E2 -9392.296} C_VEL
LIN {X 0,Y 432.339,Z 254.252,A -85,B 0,C 180,E1 -9394.678,E2 -9394.678} C_VEL
LIN {X 0,Y 432.346,Z 254.254,A -85,B 0,C 180,E1 -9398.15,E2 -9398.15} C_VEL
LIN {X 0,Y 432.332,Z 254.259,A -85,B 0,C 180,E1 -9401.603,E2 -9401.603} C_VEL
LIN {X 0,Y 432.333,Z 254.253,A -85,B 0,C 180,E1 -9404.348,E2 -9404.348} C_VEL
LIN {X 0,Y 432.32,Z 254.255,A -85,B 0,C 180,E1 -9407.017,E2 -9407.017} C_VEL
LIN {X 0,Y 432.334,Z 254.257,A -85,B 0,C 180,E1 -9409.822,E2 -9409.822} C_VEL
LIN {X 0,Y 432.306,Z 254.258,A -85,B 0,C 180,E1 -9413.023,E2 -9413.023} C_VEL
LIN {X 0,Y 432.361,Z 254.255,A -85,B 0,C 180,E1 -9415.997,E2 -9415.997} C_VEL
LIN {X 0,Y 432.349,Z 254.261,A -85,B 0,C 180,E1 -9419.49,E2 -9419.49} C_VEL
LIN {X 0,Y 432.419,Z 254.334,A -85,B 0,C 180,E1 -9421.009,E2 -9421.009} C_VEL
LIN {X 0,Y 435.969,Z 270.889,A -85,B 0,C 180,E1 -9424.199,E2 -9424.199} C_VEL
LIN {X 0,Y 436.023,Z 275.494,A -85,B 0,C 180,E1 -9425.018,E2 -9425.018} C_VEL
LIN {X 0,Y 434.946,Z 292.193,A -85,B 0,C 180,E1 -9427.9,E2 -9427.9} C_VEL
LIN {X 0,Y 439.645,Z 319.752,A -85,B 0,C 180,E1 -9428.593,E2 -9428.593} C_VEL
LIN {X 0,Y 438.209,Z 430.503,A -85,B 0,C 180,E1 -9430.44,E2 -9430.44} C_VEL
LIN {X 0,Y 437.633,Z 445.095,A -85,B 0,C 180,E1 -9430.871,E2 -9430.871} C_VEL
LIN {X 0,Y 436.987,Z 459.239,A -85,B 0,C 180,E1 -9431.488,E2 -9431.488} C_VEL
LIN {X 0,Y 436.321,Z 471.221,A -85,B 0,C 180,E1 -9432.18,E2 -9432.18} C_VEL
LIN {X 0,Y 435.434,Z 484.017,A -85,B 0,C 180,E1 -9433.111,E2 -9433.111} C_VEL
LIN {X 0,Y 434.638,Z 495.661,A -85,B 0,C 180,E1 -9434.165,E2 -9434.165} C_VEL
LIN {X 0,Y 433.818,Z 505.339,A -85,B 0,C 180,E1 -9435.217,E2 -9435.217} C_VEL
LIN {X 0,Y 433.079,Z 516.09,A -85,B 0,C 180,E1 -9436.63,E2 -9436.63} C_VEL
LIN {X 0,Y 432.461,Z 524.955,A -85,B 0,C 180,E1 -9438.042,E2 -9438.042} C_VEL
LIN {X 0,Y 431.964,Z 532.318,A -85,B 0,C 180,E1 -9439.453,E2 -9439.453} C_VEL
LIN {X 0,Y 431.601,Z 539.362,A -85,B 0,C 180,E1 -9441.101,E2 -9441.101} C_VEL
LIN {X 0,Y 431.391,Z 545.678,A -85,B 0,C 180,E1 -9442.982,E2 -9442.982} C_VEL
LIN {X 0,Y 431.265,Z 549.269,A -85,B 0,C 180,E1 -9444.389,E2 -9444.389} C_VEL
LIN {X 0,Y 431.16,Z 552.782,A -85,B 0,C 180,E1 -9446.262,E2 -9446.262} C_VEL
LIN {X 0,Y 431.201,Z 554.888,A -85,B 0,C 180,E1 -9448.132,E2 -9448.132} C_VEL
LIN {X 0,Y 431.167,Z 555.637,A -85,B 0,C 180,E1 -9450,E2 -9450} C_VEL
LIN {X 0,Y 431.201,Z 555.052,A -85,B 0,C 180,E1 -9451.868,E2 -9451.868} C_VEL
LIN {X 0,Y 431.159,Z 553.118,A -85,B 0,C 180,E1 -9453.738,E2 -9453.738} C_VEL
LIN {X 0,Y 431.278,Z 549.786,A -85,B 0,C 180,E1 -9455.611,E2 -9455.611} C_VEL
LIN {X 0,Y 431.415,Z 544.962,A -85,B 0,C 180,E1 -9457.488,E2 -9457.488} C_VEL
LIN {X 0,Y 431.742,Z 538.515,A -85,B 0,C 180,E1 -9459.368,E2 -9459.368} C_VEL
LIN {X 0,Y 432.226,Z 531.356,A -85,B 0,C 180,E1 -9461.014,E2 -9461.014} C_VEL
LIN {X 0,Y 432.793,Z 523.995,A -85,B 0,C 180,E1 -9462.404,E2 -9462.404} C_VEL
LIN {X 0,Y 433.449,Z 515.087,A -85,B 0,C 180,E1 -9463.813,E2 -9463.813} C_VEL
LIN {X 0,Y 434.18,Z 506.056,A -85,B 0,C 180,E1 -9465.01,E2 -9465.01} C_VEL
LIN {X 0,Y 435.133,Z 495.505,A -85,B 0,C 180,E1 -9466.177,E2 -9466.177} C_VEL
LIN {X 0,Y 436.082,Z 484.032,A -85,B 0,C 180,E1 -9467.225,E2 -9467.225} C_VEL
LIN {X 0,Y 436.881,Z 472.458,A -85,B 0,C 180,E1 -9468.092,E2 -9468.092} C_VEL
LIN {X 0,Y 437.844,Z 458.53,A -85,B 0,C 180,E1 -9468.907,E2 -9468.907} C_VEL
LIN {X 0,Y 438.566,Z 445.411,A -85,B 0,C 180,E1 -9469.482,E2 -9469.482} C_VEL
LIN {X 0,Y 439.164,Z 431.329,A -85,B 0,C 180,E1 -9469.911,E2 -9469.911} C_VEL
LIN {X 0,Y 439.725,Z 400.073,A -85,B 0,C 180,E1 -9470.464,E2 -9470.464} C_VEL
LIN {X 0,Y 440.778,Z 319.064,A -85,B 0,C 180,E1 -9471.825,E2 -9471.825} C_VEL
LIN {X 0,Y 436.973,Z 298.474,A -85,B 0,C 180,E1 -9472.417,E2 -9472.417} C_VEL
LIN {X 0,Y 435.584,Z 291.799,A -85,B 0,C 180,E1 -9472.64,E2 -9472.64} C_VEL
LIN {X 0,Y 436.857,Z 275.483,A -85,B 0,C 180,E1 -9475.544,E2 -9475.544} C_VEL
LIN {X 0,Y 436.117,Z 270.257,A -85,B 0,C 180,E1 -9476.563,E2 -9476.563} C_VEL
LIN {X 0,Y 433.288,Z 257.943,A -85,B 0,C 180,E1 -9479.117,E2 -9479.117} C_VEL
LIN {X 0,Y 432.367,Z 254.255,A -85,B 0,C 180,E1 -9479.921,E2 -9479.921} C_VEL
LIN {X 0,Y 432.34,Z 254.262,A -85,B 0,C 180,E1 -9483.551,E2 -9483.551} C_VEL
LIN {X 0,Y 432.338,Z 254.261,A -85,B 0,C 180,E1 -9485.817,E2 -9485.817} C_VEL
LIN {X 0,Y 432.346,Z 254.258,A -85,B 0,C 180,E1 -9489.342,E2 -9489.342} C_VEL
LIN {X 0,Y 432.369,Z 254.249,A -85,B 0,C 180,E1 -9491.792,E2 -9491.792} C_VEL
LIN {X 0,Y 432.377,Z 254.255,A -85,B 0,C 180,E1 -9494.34,E2 -9494.34} C_VEL
LIN {X 0,Y 432.331,Z 254.258,A -85,B 0,C 180,E1 -9498.202,E2 -9498.202} C_VEL
LIN {X 0,Y 432.34,Z 254.254,A -85,B 0,C 180,E1 -9501.284,E2 -9501.284} C_VEL
LIN {X 0,Y 432.342,Z 254.241,A -85,B 0,C 180,E1 -9504.367,E2 -9504.367} C_VEL
LIN {X 0,Y 432.32,Z 254.258,A -85,B 0,C 180,E1 -9507.556,E2 -9507.556} C_VEL
LIN {X 0,Y 432.39,Z 254.247,A -85,B 0,C 180,E1 -9509.743,E2 -9509.743} C_VEL
LIN {X 0,Y 432.394,Z 254.245,A -85,B 0,C 180,E1 -9513.371,E2 -9513.371} C_VEL
LIN {X 0,Y 432.366,Z 254.25,A -85,B 0,C 180,E1 -9516.022,E2 -9516.022} C_VEL
LIN {X 0,Y 432.344,Z 254.252,A -85,B 0,C 180,E1 -9519.045,E2 -9519.045} C_VEL
LIN {X 0,Y 432.372,Z 254.252,A -85,B 0,C 180,E1 -9522.01,E2 -9522.01} C_VEL
LIN {X 0,Y 432.388,Z 254.244,A -85,B 0,C 180,E1 -9524.925,E2 -9524.925} C_VEL
LIN {X 0,Y 432.452,Z 254.236,A -85,B 0,C 180,E1 -9527.802,E2 -9527.802} C_VEL
LIN {X 0,Y 432.484,Z 254.235,A -85,B 0,C 180,E1 -9531.589,E2 -9531.589} C_VEL
LIN {X 0,Y 432.589,Z 254.222,A -85,B 0,C 180,E1 -9534.405,E2 -9534.405} C_VEL
LIN {X 0,Y 432.597,Z 254.22,A -85,B 0,C 180,E1 -9538.137,E2 -9538.137} C_VEL
LIN {X 0,Y 432.725,Z 254.204,A -85,B 0,C 180,E1 -9539.999,E2 -9539.999} C_VEL
LIN {X 0,Y 432.596,Z 254.221,A -85,B 0,C 180,E1 -9542.792,E2 -9542.792} C_VEL
LIN {X 0,Y 432.562,Z 254.223,A -85,B 0,C 180,E1 -9546.529,E2 -9546.529} C_VEL
LIN {X 0,Y 432.433,Z 254.24,A -85,B 0,C 180,E1 -9549.352,E2 -9549.352} C_VEL
LIN {X 0,Y 432.419,Z 254.247,A -85,B 0,C 180,E1 -9552.802,E2 -9552.802} C_VEL
LIN {X 0,Y 432.4,Z 254.248,A -85,B 0,C 180,E1 -9556.478,E2 -9556.478} C_VEL
LIN {X 0,Y 432.367,Z 254.249,A -85,B 0,C 180,E1 -9559.957,E2 -9559.957} C_VEL
LIN {X 0,Y 432.312,Z 254.259,A -85,B 0,C 180,E1 -9562.963,E2 -9562.963} C_VEL
LIN {X 0,Y 432.351,Z 254.253,A -85,B 0,C 180,E1 -9566.032,E2 -9566.032} C_VEL
LIN {X 0,Y 432.338,Z 254.251,A -85,B 0,C 180,E1 -9569.186,E2 -9569.186} C_VEL
LIN {X 0,Y 432.311,Z 254.256,A -85,B 0,C 180,E1 -9572.292,E2 -9572.292} C_VEL
LIN {X 0,Y 432.326,Z 254.25,A -85,B 0,C 180,E1 -9574.676,E2 -9574.676} C_VEL
LIN {X 0,Y 432.338,Z 254.256,A -85,B 0,C 180,E1 -9578.148,E2 -9578.148} C_VEL
LIN {X 0,Y 432.359,Z 254.252,A -85,B 0,C 180,E1 -9581.607,E2 -9581.607} C_VEL
LIN {X 0,Y 432.364,Z 254.255,A -85,B 0,C 180,E1 -9584.341,E2 -9584.341} C_VEL
LIN {X 0,Y 432.351,Z 254.255,A -85,B 0,C 180,E1 -9587.009,E2 -9587.009} C_VEL
LIN {X 0,Y 432.391,Z 254.373,A -85,B 0,C 180,E1 -9589.735,E2 -9589.735} C_VEL
LIN {X 0,Y 435.247,Z 267.28,A -85,B 0,C 180,E1 -9592.735,E2 -9592.735} C_VEL
LIN {X 0,Y 435.837,Z 270.61,A -85,B 0,C 180,E1 -9593.447,E2 -9593.447} C_VEL
LIN {X 0,Y 439.7,Z 285.813,A -85,B 0,C 180,E1 -9593.957,E2 -9593.957} C_VEL
LIN {X 0,Y 441.171,Z 293.097,A -85,B 0,C 180,E1 -9594.174,E2 -9594.174} C_VEL
LIN {X 0,Y 439.444,Z 406.93,A -85,B 0,C 180,E1 -9596.1,E2 -9596.1} C_VEL
LIN {X 0,Y 438.96,Z 421.485,A -85,B 0,C 180,E1 -9596.535,E2 -9596.535} C_VEL
LIN {X 0,Y 438.3,Z 434.569,A -85,B 0,C 180,E1 -9597.101,E2 -9597.101} C_VEL
LIN {X 0,Y 437.523,Z 447.622,A -85,B 0,C 180,E1 -9597.854,E2 -9597.854} C_VEL
LIN {X 0,Y 436.583,Z 460.974,A -85,B 0,C 180,E1 -9598.845,E2 -9598.845} C_VEL
LIN {X 0,Y 435.568,Z 473.284,A -85,B 0,C 180,E1 -9599.988,E2 -9599.988} C_VEL
LIN {X 0,Y 434.625,Z 484.291,A -85,B 0,C 180,E1 -9601.246,E2 -9601.246} C_VEL
LIN {X 0,Y 433.856,Z 493.398,A -85,B 0,C 180,E1 -9602.506,E2 -9602.506} C_VEL
LIN {X 0,Y 433.116,Z 502.482,A -85,B 0,C 180,E1 -9604.017,E2 -9604.017} C_VEL
LIN {X 0,Y 432.504,Z 509.806,A -85,B 0,C 180,E1 -9605.497,E2 -9605.497} C_VEL
LIN {X 0,Y 432.029,Z 515.986,A -85,B 0,C 180,E1 -9607.02,E2 -9607.02} C_VEL
LIN {X 0,Y 431.74,Z 520.079,A -85,B 0,C 180,E1 -9608.242,E2 -9608.242} C_VEL
LIN {X 0,Y 430.917,Z 522.252,A -85,B 0,C 180,E1 -9608.967,E2 -9608.967} C_VEL
LIN {X 0,Y 427.858,Z 525.374,A -85,B 0,C 180,E1 -9610.156,E2 -9610.156} C_VEL
LIN {X 0,Y 425.321,Z 527.456,A -85,B 0,C 180,E1 -9611.133,E2 -9611.133} C_VEL
LIN {X 0,Y 424.202,Z 528.737,A -85,B 0,C 180,E1 -9611.9,E2 -9611.9} C_VEL
LIN {X 0,Y 424.092,Z 529.06,A -85,B 0,C 180,E1 -9612.162,E2 -9612.162} C_VEL
LIN {X 0,Y 424.046,Z 530.995,A -85,B 0,C 180,E1 -9613.995,E2 -9613.995} C_VEL
LIN {X 0,Y 423.96,Z 531.595,A -85,B 0,C 180,E1 -9615.602,E2 -9615.602} C_VEL
LIN {X 0,Y 424.033,Z 531.095,A -85,B 0,C 180,E1 -9617.558,E2 -9617.558} C_VEL
LIN {X 0,Y 424.069,Z 529.223,A -85,B 0,C 180,E1 -9619.497,E2 -9619.497} C_VEL
LIN {X 0,Y 424.259,Z 525.921,A -85,B 0,C 180,E1 -9621.426,E2 -9621.426} C_VEL
LIN {X 0,Y 424.5,Z 521.035,A -85,B 0,C 180,E1 -9623.375,E2 -9623.375} C_VEL
LIN {X 0,Y 424.836,Z 514.706,A -85,B 0,C 180,E1 -9625.256,E2 -9625.256} C_VEL
LIN {X 0,Y 425.32,Z 507.577,A -85,B 0,C 180,E1 -9626.922,E2 -9626.922} C_VEL
LIN {X 0,Y 425.898,Z 500.127,A -85,B 0,C 180,E1 -9628.345,E2 -9628.345} C_VEL
LIN {X 0,Y 426.603,Z 491.2,A -85,B 0,C 180,E1 -9629.764,E2 -9629.764} C_VEL
LIN {X 0,Y 427.505,Z 480.405,A -85,B 0,C 180,E1 -9631.178,E2 -9631.178} C_VEL
LIN {X 0,Y 428.402,Z 469.461,A -85,B 0,C 180,E1 -9632.351,E2 -9632.351} C_VEL
LIN {X 0,Y 429.262,Z 457.478,A -85,B 0,C 180,E1 -9633.403,E2 -9633.403} C_VEL
LIN {X 0,Y 430.046,Z 444.693,A -85,B 0,C 180,E1 -9634.3,E2 -9634.3} C_VEL
LIN {X 0,Y 430.706,Z 431.532,A -85,B 0,C 180,E1 -9635.017,E2 -9635.017} C_VEL
LIN {X 0,Y 431.262,Z 417.041,A -85,B 0,C 180,E1 -9635.592,E2 -9635.592} C_VEL
LIN {X 0,Y 431.633,Z 402.923,A -85,B 0,C 180,E1 -9635.958,E2 -9635.958} C_VEL
LIN {X 0,Y 433.099,Z 293.087,A -85,B 0,C 180,E1 -9637.805,E2 -9637.805} C_VEL
LIN {X 0,Y 428.206,Z 270.285,A -85,B 0,C 180,E1 -9638.447,E2 -9638.447} C_VEL
LIN {X 0,Y 427.508,Z 265.437,A -85,B 0,C 180,E1 -9639.484,E2 -9639.484} C_VEL
LIN {X 0,Y 425.431,Z 255.12,A -85,B 0,C 180,E1 -9641.796,E2 -9641.796} C_VEL
LIN {X 0,Y 425.336,Z 255.132,A -85,B 0,C 180,E1 -9645.33,E2 -9645.33} C_VEL
LIN {X 0,Y 425.319,Z 255.128,A -85,B 0,C 180,E1 -9648.298,E2 -9648.298} C_VEL
LIN {X 0,Y 425.279,Z 255.134,A -85,B 0,C 180,E1 -9651.319,E2 -9651.319} C_VEL
LIN {X 0,Y 425.315,Z 255.127,A -85,B 0,C 180,E1 -9654.66,E2 -9654.66} C_VEL
LIN {X 0,Y 425.337,Z 255.131,A -85,B 0,C 180,E1 -9657.558,E2 -9657.558} C_VEL
LIN {X 0,Y 425.287,Z 255.131,A -85,B 0,C 180,E1 -9660.815,E2 -9660.815} C_VEL
LIN {X 0,Y 425.298,Z 255.129,A -85,B 0,C 180,E1 -9664.289,E2 -9664.289} C_VEL
LIN {X 0,Y 425.275,Z 255.136,A -85,B 0,C 180,E1 -9667.694,E2 -9667.694} C_VEL
LIN {X 0,Y 425.29,Z 255.13,A -85,B 0,C 180,E1 -9670.525,E2 -9670.525} C_VEL
LIN {X 0,Y 425.319,Z 255.134,A -85,B 0,C 180,E1 -9673.362,E2 -9673.362} C_VEL
LIN {X 0,Y 425.303,Z 255.129,A -85,B 0,C 180,E1 -9676.641,E2 -9676.641} C_VEL
LIN {X 0,Y 425.298,Z 255.13,A -85,B 0,C 180,E1 -9679.876,E2 -9679.876} C_VEL
LIN {X 0,Y 425.274,Z 255.133,A -85,B 0,C 180,E1 -9682.488,E2 -9682.488} C_VEL
LIN {X 0,Y 425.295,Z 255.13,A -85,B 0,C 180,E1 -9685.818,E2 -9685.818} C_VEL
LIN {X 0,Y 425.288,Z 255.135,A -85,B 0,C 180,E1 -9689.238,E2 -9689.238} C_VEL
LIN {X 0,Y 425.339,Z 255.125,A -85,B 0,C 180,E1 -9692.443,E2 -9692.443} C_VEL
LIN {X 0,Y 425.34,Z 255.124,A -85,B 0,C 180,E1 -9695.603,E2 -9695.603} C_VEL
LIN {X 0,Y 425.282,Z 255.136,A -85,B 0,C 180,E1 -9698.683,E2 -9698.683} C_VEL
LIN {X 0,Y 425.322,Z 255.126,A -85,B 0,C 180,E1 -9701.704,E2 -9701.704} C_VEL
LIN {X 0,Y 425.339,Z 255.13,A -85,B 0,C 180,E1 -9704.672,E2 -9704.672} C_VEL
LIN {X 0,Y 425.402,Z 255.116,A -85,B 0,C 180,E1 -9707.599,E2 -9707.599} C_VEL
LIN {X 0,Y 425.433,Z 255.112,A -85,B 0,C 180,E1 -9711.451,E2 -9711.451} C_VEL
LIN {X 0,Y 425.548,Z 255.102,A -85,B 0,C 180,E1 -9714.315,E2 -9714.315} C_VEL
LIN {X 0,Y 425.568,Z 255.098,A -85,B 0,C 180,E1 -9718.109,E2 -9718.109} C_VEL
LIN {X 0,Y 425.695,Z 255.081,A -85,B 0,C 180,E1 -9720.001,E2 -9720.001} C_VEL
LIN {X 0,Y 425.55,Z 255.1,A -85,B 0,C 180,E1 -9722.841,E2 -9722.841} C_VEL
LIN {X 0,Y 425.523,Z 255.105,A -85,B 0,C 180,E1 -9726.64,E2 -9726.64} C_VEL
LIN {X 0,Y 425.395,Z 255.117,A -85,B 0,C 180,E1 -9729.511,E2 -9729.511} C_VEL
LIN {X 0,Y 425.388,Z 255.119,A -85,B 0,C 180,E1 -9732.905,E2 -9732.905} C_VEL
LIN {X 0,Y 425.365,Z 255.123,A -85,B 0,C 180,E1 -9736.61,E2 -9736.61} C_VEL
LIN {X 0,Y 425.324,Z 255.128,A -85,B 0,C 180,E1 -9739.637,E2 -9739.637} C_VEL
LIN {X 0,Y 425.284,Z 255.135,A -85,B 0,C 180,E1 -9742.34,E2 -9742.34} C_VEL
LIN {X 0,Y 425.292,Z 255.131,A -85,B 0,C 180,E1 -9745.447,E2 -9745.447} C_VEL
LIN {X 0,Y 425.335,Z 255.125,A -85,B 0,C 180,E1 -9748.633,E2 -9748.633} C_VEL
LIN {X 0,Y 425.27,Z 255.14,A -85,B 0,C 180,E1 -9751.927,E2 -9751.927} C_VEL
LIN {X 0,Y 425.298,Z 255.131,A -85,B 0,C 180,E1 -9755.337,E2 -9755.337} C_VEL
LIN {X 0,Y 425.302,Z 255.129,A -85,B 0,C 180,E1 -9759.045,E2 -9759.045} C_VEL
LIN {X 0,Y 425.274,Z 255.132,A -85,B 0,C 180,E1 -9762.654,E2 -9762.654} C_VEL
LIN {X 0,Y 425.261,Z 255.136,A -85,B 0,C 180,E1 -9766.045,E2 -9766.045} C_VEL
LIN {X 0,Y 425.274,Z 255.132,A -85,B 0,C 180,E1 -9768.622,E2 -9768.622} C_VEL
LIN {X 0,Y 425.293,Z 255.132,A -85,B 0,C 180,E1 -9771.102,E2 -9771.102} C_VEL
LIN {X 0,Y 425.3,Z 255.129,A -85,B 0,C 180,E1 -9774.665,E2 -9774.665} C_VEL
LIN {X 0,Y 425.267,Z 255.142,A -85,B 0,C 180,E1 -9778.074,E2 -9778.074} C_VEL
LIN {X 0,Y 425.33,Z 255.186,A -85,B 0,C 180,E1 -9780.736,E2 -9780.736} C_VEL
LIN {X 0,Y 428.641,Z 270.391,A -85,B 0,C 180,E1 -9783.725,E2 -9783.725} C_VEL
LIN {X 0,Y 429.212,Z 275.074,A -85,B 0,C 180,E1 -9784.602,E2 -9784.602} C_VEL
LIN {X 0,Y 428.074,Z 291.939,A -85,B 0,C 180,E1 -9787.561,E2 -9787.561} C_VEL
LIN {X 0,Y 432.922,Z 320.305,A -85,B 0,C 180,E1 -9788.297,E2 -9788.297} C_VEL
LIN {X 0,Y 431.44,Z 429.94,A -85,B 0,C 180,E1 -9790.152,E2 -9790.152} C_VEL
LIN {X 0,Y 430.872,Z 444.662,A -85,B 0,C 180,E1 -9790.59,E2 -9790.59} C_VEL
LIN {X 0,Y 430.151,Z 458.942,A -85,B 0,C 180,E1 -9791.218,E2 -9791.218} C_VEL
LIN {X 0,Y 429.382,Z 472.217,A -85,B 0,C 180,E1 -9792.005,E2 -9792.005} C_VEL
LIN {X 0,Y 428.479,Z 484.79,A -85,B 0,C 180,E1 -9792.951,E2 -9792.951} C_VEL
LIN {X 0,Y 427.661,Z 496.277,A -85,B 0,C 180,E1 -9794.023,E2 -9794.023} C_VEL
LIN {X 0,Y 426.744,Z 506.813,A -85,B 0,C 180,E1 -9795.211,E2 -9795.211} C_VEL
LIN {X 0,Y 425.977,Z 517.295,A -85,B 0,C 180,E1 -9796.645,E2 -9796.645} C_VEL
LIN {X 0,Y 425.401,Z 525.935,A -85,B 0,C 180,E1 -9798.082,E2 -9798.082} C_VEL
LIN {X 0,Y 424.789,Z 534.17,A -85,B 0,C 180,E1 -9799.755,E2 -9799.755} C_VEL
LIN {X 0,Y 424.456,Z 540.798,A -85,B 0,C 180,E1 -9801.43,E2 -9801.43} C_VEL
LIN {X 0,Y 424.249,Z 546.671,A -85,B 0,C 180,E1 -9803.341,E2 -9803.341} C_VEL
LIN {X 0,Y 424.168,Z 550.951,A -85,B 0,C 180,E1 -9805.248,E2 -9805.248} C_VEL
LIN {X 0,Y 424.122,Z 553.772,A -85,B 0,C 180,E1 -9807.15,E2 -9807.15} C_VEL
LIN {X 0,Y 424.088,Z 555.215,A -85,B 0,C 180,E1 -9809.05,E2 -9809.05} C_VEL
LIN {X 0,Y 424.088,Z 555.316,A -85,B 0,C 180,E1 -9810.949,E2 -9810.949} C_VEL
LIN {X 0,Y 424.119,Z 554.084,A -85,B 0,C 180,E1 -9812.849,E2 -9812.849} C_VEL
LIN {X 0,Y 424.171,Z 551.488,A -85,B 0,C 180,E1 -9814.752,E2 -9814.752} C_VEL
LIN {X 0,Y 424.252,Z 547.445,A -85,B 0,C 180,E1 -9816.659,E2 -9816.659} C_VEL
LIN {X 0,Y 424.498,Z 541.858,A -85,B 0,C 180,E1 -9818.569,E2 -9818.569} C_VEL
LIN {X 0,Y 424.862,Z 535.573,A -85,B 0,C 180,E1 -9820.243,E2 -9820.243} C_VEL
LIN {X 0,Y 425.552,Z 527.767,A -85,B 0,C 180,E1 -9821.913,E2 -9821.913} C_VEL
LIN {X 0,Y 426.126,Z 519.634,A -85,B 0,C 180,E1 -9823.35,E2 -9823.35} C_VEL
LIN {X 0,Y 426.97,Z 509.857,A -85,B 0,C 180,E1 -9824.781,E2 -9824.781} C_VEL
LIN {X 0,Y 427.956,Z 499.022,A -85,B 0,C 180,E1 -9826.088,E2 -9826.088} C_VEL
LIN {X 0,Y 429.101,Z 487.033,A -85,B 0,C 180,E1 -9827.269,E2 -9827.269} C_VEL
LIN {X 0,Y 430.043,Z 474.997,A -85,B 0,C 180,E1 -9828.232,E2 -9828.232} C_VEL
LIN {X 0,Y 431.018,Z 461.275,A -85,B 0,C 180,E1 -9829.094,E2 -9829.094} C_VEL
LIN {X 0,Y 431.84,Z 447.688,A -85,B 0,C 180,E1 -9829.736,E2 -9829.736} C_VEL
LIN {X 0,Y 432.472,Z 433.732,A -85,B 0,C 180,E1 -9830.201,E2 -9830.201} C_VEL
LIN {X 0,Y 432.923,Z 416.284,A -85,B 0,C 180,E1 -9830.551,E2 -9830.551} C_VEL
LIN {X 0,Y 434.242,Z 319.439,A -85,B 0,C 180,E1 -9832.207,E2 -9832.207} C_VEL
LIN {X 0,Y 430.301,Z 298.58,A -85,B 0,C 180,E1 -9832.827,E2 -9832.827} C_VEL
LIN {X 0,Y 428.833,Z 291.613,A -85,B 0,C 180,E1 -9833.063,E2 -9833.063} C_VEL
LIN {X 0,Y 430.027,Z 276.575,A -85,B 0,C 180,E1 -9835.788,E2 -9835.788} C_VEL
LIN {X 0,Y 428.357,Z 267.565,A -85,B 0,C 180,E1 -9837.628,E2 -9837.628} C_VEL
LIN {X 0,Y 425.327,Z 255.132,A -85,B 0,C 180,E1 -9840.324,E2 -9840.324} C_VEL
LIN {X 0,Y 425.283,Z 255.14,A -85,B 0,C 180,E1 -9843.047,E2 -9843.047} C_VEL
LIN {X 0,Y 425.282,Z 255.141,A -85,B 0,C 180,E1 -9845.927,E2 -9845.927} C_VEL
LIN {X 0,Y 425.293,Z 255.137,A -85,B 0,C 180,E1 -9849.041,E2 -9849.041} C_VEL
LIN {X 0,Y 425.33,Z 255.131,A -85,B 0,C 180,E1 -9852.645,E2 -9852.645} C_VEL
LIN {X 0,Y 425.293,Z 255.131,A -85,B 0,C 180,E1 -9855.28,E2 -9855.28} C_VEL
LIN {X 0,Y 425.272,Z 255.137,A -85,B 0,C 180,E1 -9858.62,E2 -9858.62} C_VEL
LIN {X 0,Y 425.304,Z 255.13,A -85,B 0,C 180,E1 -9861.101,E2 -9861.101} C_VEL
LIN {X 0,Y 425.297,Z 255.118,A -85,B 0,C 180,E1 -9864.663,E2 -9864.663} C_VEL
LIN {X 0,Y 425.263,Z 255.136,A -85,B 0,C 180,E1 -9868.072,E2 -9868.072} C_VEL
LIN {X 0,Y 425.333,Z 255.127,A -85,B 0,C 180,E1 -9871.367,E2 -9871.367} C_VEL
LIN {X 0,Y 425.29,Z 255.131,A -85,B 0,C 180,E1 -9874.553,E2 -9874.553} C_VEL
LIN {X 0,Y 425.282,Z 255.136,A -85,B 0,C 180,E1 -9877.66,E2 -9877.66} C_VEL
LIN {X 0,Y 425.356,Z 255.121,A -85,B 0,C 180,E1 -9880.703,E2 -9880.703} C_VEL
LIN {X 0,Y 425.382,Z 255.119,A -85,B 0,C 180,E1 -9883.687,E2 -9883.687} C_VEL
LIN {X 0,Y 425.405,Z 255.116,A -85,B 0,C 180,E1 -9887.597,E2 -9887.597} C_VEL
LIN {X 0,Y 425.435,Z 255.115,A -85,B 0,C 180,E1 -9891.449,E2 -9891.449} C_VEL
LIN {X 0,Y 425.546,Z 255.099,A -85,B 0,C 180,E1 -9894.312,E2 -9894.312} C_VEL
LIN {X 0,Y 425.567,Z 255.096,A -85,B 0,C 180,E1 -9898.106,E2 -9898.106} C_VEL
LIN {X 0,Y 425.695,Z 255.08,A -85,B 0,C 180,E1 -9899.999,E2 -9899.999} C_VEL
LIN {X 0,Y 425.548,Z 255.1,A -85,B 0,C 180,E1 -9902.839,E2 -9902.839} C_VEL
LIN {X 0,Y 425.518,Z 255.101,A -85,B 0,C 180,E1 -9906.658,E2 -9906.658} C_VEL
LIN {X 0,Y 425.391,Z 255.116,A -85,B 0,C 180,E1 -9909.508,E2 -9909.508} C_VEL
LIN {X 0,Y 425.382,Z 255.122,A -85,B 0,C 180,E1 -9912.903,E2 -9912.903} C_VEL
LIN {X 0,Y 425.349,Z 255.127,A -85,B 0,C 180,E1 -9916.604,E2 -9916.604} C_VEL
LIN {X 0,Y 425.35,Z 255.123,A -85,B 0,C 180,E1 -9919.647,E2 -9919.647} C_VEL
LIN {X 0,Y 425.297,Z 255.128,A -85,B 0,C 180,E1 -9923.364,E2 -9923.364} C_VEL
LIN {X 0,Y 425.334,Z 255.128,A -85,B 0,C 180,E1 -9926.843,E2 -9926.843} C_VEL
LIN {X 0,Y 425.304,Z 255.126,A -85,B 0,C 180,E1 -9929.717,E2 -9929.717} C_VEL
LIN {X 0,Y 425.268,Z 255.137,A -85,B 0,C 180,E1 -9933.047,E2 -9933.047} C_VEL
LIN {X 0,Y 425.27,Z 255.129,A -85,B 0,C 180,E1 -9935.928,E2 -9935.928} C_VEL
LIN {X 0,Y 425.298,Z 255.127,A -85,B 0,C 180,E1 -9939.045,E2 -9939.045} C_VEL
LIN {X 0,Y 425.317,Z 255.129,A -85,B 0,C 180,E1 -9942.645,E2 -9942.645} C_VEL
LIN {X 0,Y 425.32,Z 255.133,A -85,B 0,C 180,E1 -9946.053,E2 -9946.053} C_VEL
LIN {X 0,Y 425.332,Z 255.258,A -85,B 0,C 180,E1 -9949.352,E2 -9949.352} C_VEL
LIN {X 0,Y 427.626,Z 265.371,A -85,B 0,C 180,E1 -9951.765,E2 -9951.765} C_VEL
LIN {X 0,Y 428.681,Z 270.606,A -85,B 0,C 180,E1 -9952.976,E2 -9952.976} C_VEL
LIN {X 0,Y 430.923,Z 277.102,A -85,B 0,C 180,E1 -9953.254,E2 -9953.254} C_VEL
LIN {X 0,Y 434.744,Z 293.969,A -85,B 0,C 180,E1 -9953.8,E2 -9953.8} C_VEL
LIN {X 0,Y 432.897,Z 407.635,A -85,B 0,C 180,E1 -9955.756,E2 -9955.756} C_VEL
LIN {X 0,Y 432.368,Z 421.784,A -85,B 0,C 180,E1 -9956.188,E2 -9956.188} C_VEL
LIN {X 0,Y 431.629,Z 435.668,A -85,B 0,C 180,E1 -9956.805,E2 -9956.805} C_VEL
LIN {X 0,Y 430.838,Z 448.164,A -85,B 0,C 180,E1 -9957.546,E2 -9957.546} C_VEL
LIN {X 0,Y 429.943,Z 460.367,A -85,B 0,C 180,E1 -9958.462,E2 -9958.462} C_VEL
LIN {X 0,Y 428.863,Z 472.672,A -85,B 0,C 180,E1 -9959.606,E2 -9959.606} C_VEL
LIN {X 0,Y 427.885,Z 483.824,A -85,B 0,C 180,E1 -9960.884,E2 -9960.884} C_VEL
LIN {X 0,Y 426.958,Z 493.9,A -85,B 0,C 180,E1 -9962.29,E2 -9962.29} C_VEL
LIN {X 0,Y 426.159,Z 502.917,A -85,B 0,C 180,E1 -9963.824,E2 -9963.824} C_VEL
LIN {X 0,Y 425.552,Z 509.944,A -85,B 0,C 180,E1 -9965.27,E2 -9965.27} C_VEL
LIN {X 0,Y 425.083,Z 515.399,A -85,B 0,C 180,E1 -9966.623,E2 -9966.623} C_VEL
LIN {X 0,Y 424.65,Z 520.87,A -85,B 0,C 180,E1 -9968.276,E2 -9968.276} C_VEL
LIN {X 0,Y 424.342,Z 525.613,A -85,B 0,C 180,E1 -9970.153,E2 -9970.153} C_VEL
LIN {X 0,Y 424.092,Z 529.06,A -85,B 0,C 180,E1 -9972.162,E2 -9972.162} C_VEL
LIN {X 0,Y 423.353,Z 530.095,A -85,B 0,C 180,E1 -9972.943,E2 -9972.943} C_VEL
LIN {X 0,Y 420.404,Z 531.243,A -85,B 0,C 180,E1 -9974.219,E2 -9974.219} C_VEL
LIN {X 0,Y 417.962,Z 531.716,A -85,B 0,C 180,E1 -9975.255,E2 -9975.255} C_VEL
LIN {X 0,Y 416.941,Z 531.802,A -85,B 0,C 180,E1 -9976.058,E2 -9976.058} C_VEL
LIN {X 0,Y 416.871,Z 531.754,A -85,B 0,C 180,E1 -9976.33,E2 -9976.33} C_VEL
LIN {X 0,Y 416.985,Z 530.697,A -85,B 0,C 180,E1 -9978.332,E2 -9978.332} C_VEL
LIN {X 0,Y 416.997,Z 528.27,A -85,B 0,C 180,E1 -9980.297,E2 -9980.297} C_VEL
LIN {X 0,Y 417.28,Z 524.41,A -85,B 0,C 180,E1 -9982.257,E2 -9982.257} C_VEL
LIN {X 0,Y 417.581,Z 518.98,A -85,B 0,C 180,E1 -9984.205,E2 -9984.205} C_VEL
LIN {X 0,Y 417.858,Z 513.835,A -85,B 0,C 180,E1 -9985.66,E2 -9985.66} C_VEL
LIN {X 0,Y 418.37,Z 506.446,A -85,B 0,C 180,E1 -9987.352,E2 -9987.352} C_VEL
LIN {X 0,Y 419.029,Z 498.73,A -85,B 0,C 180,E1 -9988.799,E2 -9988.799} C_VEL
LIN {X 0,Y 419.852,Z 489.46,A -85,B 0,C 180,E1 -9990.24,E2 -9990.24} C_VEL
LIN {X 0,Y 420.691,Z 479.236,A -85,B 0,C 180,E1 -9991.556,E2 -9991.556} C_VEL
LIN {X 0,Y 421.643,Z 467.969,A -85,B 0,C 180,E1 -9992.747,E2 -9992.747} C_VEL
LIN {X 0,Y 422.557,Z 455.546,A -85,B 0,C 180,E1 -9993.815,E2 -9993.815} C_VEL
LIN {X 0,Y 423.361,Z 442.926,A -85,B 0,C 180,E1 -9994.681,E2 -9994.681} C_VEL
LIN {X 0,Y 423.966,Z 430.483,A -85,B 0,C 180,E1 -9995.348,E2 -9995.348} C_VEL
LIN {X 0,Y 424.542,Z 416.177,A -85,B 0,C 180,E1 -9995.909,E2 -9995.909} C_VEL
LIN {X 0,Y 424.905,Z 402.317,A -85,B 0,C 180,E1 -9996.261,E2 -9996.261} C_VEL
LIN {X 0,Y 426.445,Z 294.241,A -85,B 0,C 180,E1 -9998.1,E2 -9998.1} C_VEL
LIN {X 0,Y 421.241,Z 270.481,A -85,B 0,C 180,E1 -9998.79,E2 -9998.79} C_VEL
LIN {X 0,Y 418.401,Z 255.997,A -85,B 0,C 180,E1 -10002.028,E2 -10002.028} C_VEL
LIN {X 0,Y 418.289,Z 256.009,A -85,B 0,C 180,E1 -10005.594,E2 -10005.594} C_VEL
LIN {X 0,Y 418.271,Z 256.004,A -85,B 0,C 180,E1 -10008.617,E2 -10008.617} C_VEL
LIN {X 0,Y 418.221,Z 256.017,A -85,B 0,C 180,E1 -10011.697,E2 -10011.697} C_VEL
LIN {X 0,Y 418.27,Z 256.005,A -85,B 0,C 180,E1 -10014.865,E2 -10014.865} C_VEL
LIN {X 0,Y 418.281,Z 256.005,A -85,B 0,C 180,E1 -10018.063,E2 -10018.063} C_VEL
LIN {X 0,Y 418.209,Z 256.017,A -85,B 0,C 180,E1 -10021.396,E2 -10021.396} C_VEL
LIN {X 0,Y 418.252,Z 256.007,A -85,B 0,C 180,E1 -10024.581,E2 -10024.581} C_VEL
LIN {X 0,Y 418.225,Z 256.013,A -85,B 0,C 180,E1 -10027.836,E2 -10027.836} C_VEL
LIN {X 0,Y 418.254,Z 256.009,A -85,B 0,C 180,E1 -10030.943,E2 -10030.943} C_VEL
LIN {X 0,Y 418.27,Z 256.007,A -85,B 0,C 180,E1 -10033.741,E2 -10033.741} C_VEL
LIN {X 0,Y 418.254,Z 256.006,A -85,B 0,C 180,E1 -10036.457,E2 -10036.457} C_VEL
LIN {X 0,Y 418.254,Z 256.012,A -85,B 0,C 180,E1 -10039.124,E2 -10039.124} C_VEL
LIN {X 0,Y 418.226,Z 256.01,A -85,B 0,C 180,E1 -10042.166,E2 -10042.166} C_VEL
LIN {X 0,Y 418.253,Z 256.01,A -85,B 0,C 180,E1 -10045.421,E2 -10045.421} C_VEL
LIN {X 0,Y 418.204,Z 256.015,A -85,B 0,C 180,E1 -10048.605,E2 -10048.605} C_VEL
LIN {X 0,Y 418.283,Z 256.003,A -85,B 0,C 180,E1 -10051.938,E2 -10051.938} C_VEL
LIN {X 0,Y 418.279,Z 256.008,A -85,B 0,C 180,E1 -10055.164,E2 -10055.164} C_VEL
LIN {X 0,Y 418.223,Z 256.012,A -85,B 0,C 180,E1 -10058.305,E2 -10058.305} C_VEL
LIN {X 0,Y 418.273,Z 256.005,A -85,B 0,C 180,E1 -10061.384,E2 -10061.384} C_VEL
LIN {X 0,Y 418.293,Z 256.005,A -85,B 0,C 180,E1 -10064.407,E2 -10064.407} C_VEL
LIN {X 0,Y 418.346,Z 255.996,A -85,B 0,C 180,E1 -10067.387,E2 -10067.387} C_VEL
LIN {X 0,Y 418.332,Z 256,A -85,B 0,C 180,E1 -10070.33,E2 -10070.33} C_VEL
LIN {X 0,Y 418.485,Z 255.979,A -85,B 0,C 180,E1 -10073.25,E2 -10073.25} C_VEL
LIN {X 0,Y 418.334,Z 255.997,A -85,B 0,C 180,E1 -10075.183,E2 -10075.183} C_VEL
LIN {X 0,Y 418.537,Z 255.973,A -85,B 0,C 180,E1 -10078.077,E2 -10078.077} C_VEL
LIN {X 0,Y 418.665,Z 255.957,A -85,B 0,C 180,E1 -10080.001,E2 -10080.001} C_VEL
LIN {X 0,Y 418.504,Z 255.978,A -85,B 0,C 180,E1 -10082.889,E2 -10082.889} C_VEL
LIN {X 0,Y 418.486,Z 255.98,A -85,B 0,C 180,E1 -10086.752,E2 -10086.752} C_VEL
LIN {X 0,Y 418.335,Z 255.997,A -85,B 0,C 180,E1 -10089.673,E2 -10089.673} C_VEL
LIN {X 0,Y 418.341,Z 255.996,A -85,B 0,C 180,E1 -10093.002,E2 -10093.002} C_VEL
LIN {X 0,Y 418.315,Z 256,A -85,B 0,C 180,E1 -10096.74,E2 -10096.74} C_VEL
LIN {X 0,Y 418.266,Z 256.008,A -85,B 0,C 180,E1 -10099.791,E2 -10099.791} C_VEL
LIN {X 0,Y 418.228,Z 256.01,A -85,B 0,C 180,E1 -10102.738,E2 -10102.738} C_VEL
LIN {X 0,Y 418.267,Z 256.011,A -85,B 0,C 180,E1 -10105.905,E2 -10105.905} C_VEL
LIN {X 0,Y 418.271,Z 256.004,A -85,B 0,C 180,E1 -10109.162,E2 -10109.162} C_VEL
LIN {X 0,Y 418.258,Z 256.006,A -85,B 0,C 180,E1 -10112.846,E2 -10112.846} C_VEL
LIN {X 0,Y 418.247,Z 256.01,A -85,B 0,C 180,E1 -10116.24,E2 -10116.24} C_VEL
LIN {X 0,Y 418.254,Z 256.013,A -85,B 0,C 180,E1 -10119.683,E2 -10119.683} C_VEL
LIN {X 0,Y 418.229,Z 256.011,A -85,B 0,C 180,E1 -10122.322,E2 -10122.322} C_VEL
LIN {X 0,Y 418.235,Z 256.01,A -85,B 0,C 180,E1 -10125.11,E2 -10125.11} C_VEL
LIN {X 0,Y 418.24,Z 256.014,A -85,B 0,C 180,E1 -10127.768,E2 -10127.768} C_VEL
LIN {X 0,Y 418.243,Z 256.008,A -85,B 0,C 180,E1 -10130.622,E2 -10130.622} C_VEL
LIN {X 0,Y 418.244,Z 256.01,A -85,B 0,C 180,E1 -10133.977,E2 -10133.977} C_VEL
LIN {X 0,Y 418.259,Z 256.01,A -85,B 0,C 180,E1 -10137.157,E2 -10137.157} C_VEL
LIN {X 0,Y 418.284,Z 256.069,A -85,B 0,C 180,E1 -10140.461,E2 -10140.461} C_VEL
LIN {X 0,Y 421.304,Z 269.879,A -85,B 0,C 180,E1 -10143.231,E2 -10143.231} C_VEL
LIN {X 0,Y 422.318,Z 275.723,A -85,B 0,C 180,E1 -10144.363,E2 -10144.363} C_VEL
LIN {X 0,Y 421.209,Z 291.802,A -85,B 0,C 180,E1 -10147.233,E2 -10147.233} C_VEL
LIN {X 0,Y 426.2,Z 321.519,A -85,B 0,C 180,E1 -10148.006,E2 -10148.006} C_VEL
LIN {X 0,Y 424.701,Z 429.349,A -85,B 0,C 180,E1 -10149.855,E2 -10149.855} C_VEL
LIN {X 0,Y 424.173,Z 443.465,A -85,B 0,C 180,E1 -10150.27,E2 -10150.27} C_VEL
LIN {X 0,Y 423.434,Z 456.6,A -85,B 0,C 180,E1 -10150.832,E2 -10150.832} C_VEL
LIN {X 0,Y 422.742,Z 469.659,A -85,B 0,C 180,E1 -10151.587,E2 -10151.587} C_VEL
LIN {X 0,Y 421.741,Z 482.68,A -85,B 0,C 180,E1 -10152.545,E2 -10152.545} C_VEL
LIN {X 0,Y 420.825,Z 494.5,A -85,B 0,C 180,E1 -10153.631,E2 -10153.631} C_VEL
LIN {X 0,Y 419.942,Z 504.317,A -85,B 0,C 180,E1 -10154.717,E2 -10154.717} C_VEL
LIN {X 0,Y 419.113,Z 515.182,A -85,B 0,C 180,E1 -10156.175,E2 -10156.175} C_VEL
LIN {X 0,Y 418.466,Z 524.144,A -85,B 0,C 180,E1 -10157.636,E2 -10157.636} C_VEL
LIN {X 0,Y 417.931,Z 531.588,A -85,B 0,C 180,E1 -10159.095,E2 -10159.095} C_VEL
LIN {X 0,Y 417.502,Z 538.7,A -85,B 0,C 180,E1 -10160.798,E2 -10160.798} C_VEL
LIN {X 0,Y 417.244,Z 545.078,A -85,B 0,C 180,E1 -10162.743,E2 -10162.743} C_VEL
LIN {X 0,Y 417.091,Z 548.722,A -85,B 0,C 180,E1 -10164.197,E2 -10164.197} C_VEL
LIN {X 0,Y 416.989,Z 552.284,A -85,B 0,C 180,E1 -10166.134,E2 -10166.134} C_VEL
LIN {X 0,Y 417.054,Z 554.436,A -85,B 0,C 180,E1 -10168.069,E2 -10168.069} C_VEL
LIN {X 0,Y 417.004,Z 555.227,A -85,B 0,C 180,E1 -10170,E2 -10170} C_VEL
LIN {X 0,Y 417.054,Z 554.685,A -85,B 0,C 180,E1 -10171.931,E2 -10171.931} C_VEL
LIN {X 0,Y 416.988,Z 552.802,A -85,B 0,C 180,E1 -10173.865,E2 -10173.865} C_VEL
LIN {X 0,Y 417.107,Z 549.531,A -85,B 0,C 180,E1 -10175.802,E2 -10175.802} C_VEL
LIN {X 0,Y 417.289,Z 544.763,A -85,B 0,C 180,E1 -10177.743,E2 -10177.743} C_VEL
LIN {X 0,Y 417.668,Z 538.378,A -85,B 0,C 180,E1 -10179.687,E2 -10179.687} C_VEL
LIN {X 0,Y 418.257,Z 531.29,A -85,B 0,C 180,E1 -10181.387,E2 -10181.387} C_VEL
LIN {X 0,Y 418.817,Z 523.607,A -85,B 0,C 180,E1 -10182.898,E2 -10182.898} C_VEL
LIN {X 0,Y 419.603,Z 515.027,A -85,B 0,C 180,E1 -10184.303,E2 -10184.303} C_VEL
LIN {X 0,Y 420.626,Z 504.322,A -85,B 0,C 180,E1 -10185.754,E2 -10185.754} C_VEL
LIN {X 0,Y 421.759,Z 493.517,A -85,B 0,C 180,E1 -10186.954,E2 -10186.954} C_VEL
LIN {X 0,Y 422.786,Z 481.727,A -85,B 0,C 180,E1 -10188.035,E2 -10188.035} C_VEL
LIN {X 0,Y 423.759,Z 469.887,A -85,B 0,C 180,E1 -10188.911,E2 -10188.911} C_VEL
LIN {X 0,Y 424.698,Z 456.291,A -85,B 0,C 180,E1 -10189.704,E2 -10189.704} C_VEL
LIN {X 0,Y 425.576,Z 442.531,A -85,B 0,C 180,E1 -10190.291,E2 -10190.291} C_VEL
LIN {X 0,Y 426.181,Z 428.176,A -85,B 0,C 180,E1 -10190.702,E2 -10190.702} C_VEL
LIN {X 0,Y 427.887,Z 321.11,A -85,B 0,C 180,E1 -10192.567,E2 -10192.567} C_VEL
LIN {X 0,Y 424.093,Z 300.646,A -85,B 0,C 180,E1 -10193.188,E2 -10193.188} C_VEL
LIN {X 0,Y 422.09,Z 291.355,A -85,B 0,C 180,E1 -10193.515,E2 -10193.515} C_VEL
LIN {X 0,Y 423.186,Z 278.925,A -85,B 0,C 180,E1 -10195.807,E2 -10195.807} C_VEL
LIN {X 0,Y 422.629,Z 274.618,A -85,B 0,C 180,E1 -10196.678,E2 -10196.678} C_VEL
LIN {X 0,Y 420.192,Z 263.709,A -85,B 0,C 180,E1 -10199.015,E2 -10199.015} C_VEL
LIN {X 0,Y 418.264,Z 256.013,A -85,B 0,C 180,E1 -10200.757,E2 -10200.757} C_VEL
LIN {X 0,Y 418.249,Z 256.018,A -85,B 0,C 180,E1 -10203.676,E2 -10203.676} C_VEL
LIN {X 0,Y 418.24,Z 256.011,A -85,B 0,C 180,E1 -10207.223,E2 -10207.223} C_VEL
LIN {X 0,Y 418.248,Z 256.015,A -85,B 0,C 180,E1 -10209.681,E2 -10209.681} C_VEL
LIN {X 0,Y 418.283,Z 256.01,A -85,B 0,C 180,E1 -10212.328,E2 -10212.328} C_VEL
LIN {X 0,Y 418.25,Z 256.009,A -85,B 0,C 180,E1 -10215.11,E2 -10215.11} C_VEL
LIN {X 0,Y 418.238,Z 256.012,A -85,B 0,C 180,E1 -10217.765,E2 -10217.765} C_VEL
LIN {X 0,Y 418.251,Z 256.011,A -85,B 0,C 180,E1 -10220.618,E2 -10220.618} C_VEL
LIN {X 0,Y 418.24,Z 255.997,A -85,B 0,C 180,E1 -10223.975,E2 -10223.975} C_VEL
LIN {X 0,Y 418.254,Z 256.008,A -85,B 0,C 180,E1 -10227.155,E2 -10227.155} C_VEL
LIN {X 0,Y 418.27,Z 256.006,A -85,B 0,C 180,E1 -10230.837,E2 -10230.837} C_VEL
LIN {X 0,Y 418.266,Z 256.01,A -85,B 0,C 180,E1 -10234.095,E2 -10234.095} C_VEL
LIN {X 0,Y 418.233,Z 256.01,A -85,B 0,C 180,E1 -10237.262,E2 -10237.262} C_VEL
LIN {X 0,Y 418.277,Z 256.003,A -85,B 0,C 180,E1 -10240.363,E2 -10240.363} C_VEL
LIN {X 0,Y 418.31,Z 256.001,A -85,B 0,C 180,E1 -10243.403,E2 -10243.403} C_VEL
LIN {X 0,Y 418.339,Z 255.998,A -85,B 0,C 180,E1 -10246.998,E2 -10246.998} C_VEL
LIN {X 0,Y 418.335,Z 255.998,A -85,B 0,C 180,E1 -10250.327,E2 -10250.327} C_VEL
LIN {X 0,Y 418.484,Z 255.976,A -85,B 0,C 180,E1 -10253.248,E2 -10253.248} C_VEL
LIN {X 0,Y 418.333,Z 256.003,A -85,B 0,C 180,E1 -10255.18,E2 -10255.18} C_VEL
LIN {X 0,Y 418.536,Z 255.972,A -85,B 0,C 180,E1 -10258.074,E2 -10258.074} C_VEL
LIN {X 0,Y 418.665,Z 255.956,A -85,B 0,C 180,E1 -10259.999,E2 -10259.999} C_VEL
LIN {X 0,Y 418.501,Z 255.978,A -85,B 0,C 180,E1 -10262.886,E2 -10262.886} C_VEL
LIN {X 0,Y 418.482,Z 255.978,A -85,B 0,C 180,E1 -10266.75,E2 -10266.75} C_VEL
LIN {X 0,Y 418.331,Z 255.994,A -85,B 0,C 180,E1 -10269.67,E2 -10269.67} C_VEL
LIN {X 0,Y 418.335,Z 255.998,A -85,B 0,C 180,E1 -10273,E2 -10273} C_VEL
LIN {X 0,Y 418.301,Z 256.004,A -85,B 0,C 180,E1 -10276.734,E2 -10276.734} C_VEL
LIN {X 0,Y 418.29,Z 256.003,A -85,B 0,C 180,E1 -10279.801,E2 -10279.801} C_VEL
LIN {X 0,Y 418.23,Z 256.016,A -85,B 0,C 180,E1 -10282.735,E2 -10282.735} C_VEL
LIN {X 0,Y 418.257,Z 256.008,A -85,B 0,C 180,E1 -10285.903,E2 -10285.903} C_VEL
LIN {X 0,Y 418.261,Z 256.005,A -85,B 0,C 180,E1 -10289.16,E2 -10289.16} C_VEL
LIN {X 0,Y 418.244,Z 256.014,A -85,B 0,C 180,E1 -10292.843,E2 -10292.843} C_VEL
LIN {X 0,Y 418.234,Z 256.008,A -85,B 0,C 180,E1 -10296.238,E2 -10296.238} C_VEL
LIN {X 0,Y 418.252,Z 256.006,A -85,B 0,C 180,E1 -10299.68,E2 -10299.68} C_VEL
LIN {X 0,Y 418.271,Z 256.005,A -85,B 0,C 180,E1 -10302.329,E2 -10302.329} C_VEL
